LIN {X -196.784,Y -213.016,Z 123.751,A 47.268,B 90.000,C 0.000} C_DIS
LIN {X -197.620,Y -212.241,Z 123.582,A 47.043,B 90.000,C 0.000} C_DIS
LIN {X -198.410,Y -211.503,Z 123.560,A 46.829,B 90.000,C 0.000} C_DIS
LIN {X -199.108,Y -210.846,Z 123.719,A 46.640,B 90.000,C 0.000} C_DIS
LIN {X -199.675,Y -210.309,Z 123.966,A 46.486,B 90.000,C 0.000} C_DIS
LIN {X -200.147,Y -209.860,Z 124.319,A 46.357,B 90.000,C 0.000} C_DIS
LIN {X -200.558,Y -209.467,Z 124.798,A 46.245,B 90.000,C 0.000} C_DIS
LIN {X -200.980,Y -209.062,Z 125.590,A 46.129,B 90.000,C 0.000} C_DIS
LIN {X -201.312,Y -208.742,Z 126.725,A 46.038,B 90.000,C 0.000} C_DIS
LIN {X -201.468,Y -208.592,Z 127.575,A 45.995,B 90.000,C 0.000} C_DIS
LIN {X -201.547,Y -208.516,Z 128.408,A 45.974,B 90.000,C 0.000} C_DIS
LIN {X -201.548,Y -208.515,Z 129.167,A 45.973,B 90.000,C 0.000} C_DIS
LIN {X -201.440,Y -208.619,Z 130.066,A 46.003,B 90.000,C 0.000} C_DIS
LIN {X -201.835,Y -208.237,Z 129.890,A 45.895,B 90.000,C 0.000} C_DIS
LIN {X -202.884,Y -207.215,Z 129.170,A 45.605,B 90.000,C 0.000} C_DIS
LIN {X -204.304,Y -205.814,Z 127.663,A 45.211,B 90.000,C 0.000} C_DIS
LIN {X -204.732,Y -205.390,Z 127.194,A 45.092,B 90.000,C 0.000} C_DIS
LIN {X -205.294,Y -204.827,Z 126.844,A 44.935,B 90.000,C 0.000} C_DIS
LIN {X -206.113,Y -204.004,Z 126.614,A 44.705,B 90.000,C 0.000} C_DIS
LIN {X -207.863,Y -202.220,Z 126.527,A 44.212,B 90.000,C 0.000} C_DIS
LIN {X -207.932,Y -202.149,Z 126.529,A 44.192,B 90.000,C 0.000} C_DIS
LIN {X -208.601,Y -201.459,Z 126.690,A 44.002,B 90.000,C 0.000} C_DIS
LIN {X -208.848,Y -201.203,Z 126.861,A 43.932,B 90.000,C 0.000} C_DIS
LIN {X -209.068,Y -200.974,Z 127.141,A 43.869,B 90.000,C 0.000} C_DIS
LIN {X -209.459,Y -200.566,Z 128.088,A 43.757,B 90.000,C 0.000} C_DIS
LIN {X -209.762,Y -200.250,Z 129.265,A 43.671,B 90.000,C 0.000} C_DIS
LIN {X -209.850,Y -200.157,Z 130.407,A 43.646,B 90.000,C 0.000} C_DIS
LIN {X -209.802,Y -200.208,Z 131.716,A 43.659,B 90.000,C 0.000} C_DIS
LIN {X -209.567,Y -200.453,Z 132.873,A 43.727,B 90.000,C 0.000} C_DIS
LIN {X -209.190,Y -200.847,Z 134.012,A 43.834,B 90.000,C 0.000} C_DIS
LIN {X -207.748,Y -199.461,Z 134.012,A 43.834,B 90.000,C 0.000} C_DIS
WAIT SEC 0.1
RET=EKI_SetBool("oxy","torchState",FALSE)
RET = EKI_Send("oxy","torchState")
LIN {X -194.764,Y -186.995,Z 134.012,A 43.834,B 90.000,C 0.000} C_DIS
LIN {X -184.230,Y -197.381,Z 120.997,A 46.974,B 90.000,C 0.000} C_DIS
LIN {X -196.512,Y -210.540,Z 120.997,A 46.974,B 90.000,C 0.000} C_DIS
LIN {X -197.877,Y -212.002,Z 120.997,A 46.974,B 90.000,C 0.000} C_DIS
WAIT SEC 1
RET=EKI_SetBool("oxy","torchState",TRUE)
RET = EKI_Send("oxy","torchState")
LIN {X -198.195,Y -211.704,Z 120.444,A 46.888,B 90.000,C 0.000} C_DIS
LIN {X -198.412,Y -211.501,Z 119.734,A 46.829,B 90.000,C 0.000} C_DIS
LIN {X -198.488,Y -211.430,Z 117.237,A 46.808,B 90.000,C 0.000} C_DIS
LIN {X -198.366,Y -211.545,Z 115.557,A 46.841,B 90.000,C 0.000} C_DIS
LIN {X -198.150,Y -211.746,Z 114.873,A 46.900,B 90.000,C 0.000} C_DIS
LIN {X -197.024,Y -212.794,Z 112.902,A 47.204,B 90.000,C 0.000} C_DIS
LIN {X -196.854,Y -212.952,Z 112.641,A 47.249,B 90.000,C 0.000} C_DIS
LIN {X -196.638,Y -213.151,Z 112.446,A 47.308,B 90.000,C 0.000} C_DIS
LIN {X -196.433,Y -213.340,Z 112.465,A 47.363,B 90.000,C 0.000} C_DIS
LIN {X -196.193,Y -213.561,Z 112.727,A 47.427,B 90.000,C 0.000} C_DIS
LIN {X -195.388,Y -214.298,Z 113.920,A 47.643,B 90.000,C 0.000} C_DIS
LIN {X -193.851,Y -215.688,Z 115.318,A 48.052,B 90.000,C 0.000} C_DIS
LIN {X -192.222,Y -217.141,Z 116.537,A 48.483,B 90.000,C 0.000} C_DIS
LIN {X -190.581,Y -218.584,Z 117.751,A 48.915,B 90.000,C 0.000} C_DIS
LIN {X -189.444,Y -219.570,Z 118.907,A 49.213,B 90.000,C 0.000} C_DIS
LIN {X -188.072,Y -220.746,Z 120.635,A 49.570,B 90.000,C 0.000} C_DIS
LIN {X -186.854,Y -221.778,Z 122.333,A 49.885,B 90.000,C 0.000} C_DIS
LIN {X -186.543,Y -222.040,Z 123.009,A 49.965,B 90.000,C 0.000} C_DIS
LIN {X -186.357,Y -222.196,Z 123.639,A 50.013,B 90.000,C 0.000} C_DIS
LIN {X -186.301,Y -222.243,Z 124.194,A 50.028,B 90.000,C 0.000} C_DIS
LIN {X -186.382,Y -222.175,Z 124.643,A 50.007,B 90.000,C 0.000} C_DIS
LIN {X -186.558,Y -222.027,Z 124.964,A 49.961,B 90.000,C 0.000} C_DIS
LIN {X -186.818,Y -221.809,Z 125.228,A 49.894,B 90.000,C 0.000} C_DIS
LIN {X -187.628,Y -221.124,Z 125.617,A 49.685,B 90.000,C 0.000} C_DIS
LIN {X -189.526,Y -219.498,Z 125.677,A 49.191,B 90.000,C 0.000} C_DIS
LIN {X -189.856,Y -219.214,Z 125.662,A 49.105,B 90.000,C 0.000} C_DIS
LIN {X -190.574,Y -218.590,Z 125.514,A 48.917,B 90.000,C 0.000} C_DIS
LIN {X -191.225,Y -218.021,Z 125.214,A 48.746,B 90.000,C 0.000} C_DIS
LIN {X -192.885,Y -216.546,Z 124.065,A 48.308,B 90.000,C 0.000} C_DIS
LIN {X -194.538,Y -215.067,Z 122.914,A 47.869,B 90.000,C 0.000} C_DIS
LIN {X -194.792,Y -214.839,Z 122.737,A 47.802,B 90.000,C 0.000} C_DIS
LIN {X -196.523,Y -213.256,Z 121.874,A 47.338,B 90.000,C 0.000} C_DIS
LIN {X -197.278,Y -212.559,Z 121.499,A 47.135,B 90.000,C 0.000} C_DIS
LIN {X -197.877,Y -212.002,Z 120.997,A 46.974,B 90.000,C 0.000} C_DIS
LIN {X -196.512,Y -210.540,Z 120.997,A 46.974,B 90.000,C 0.000} C_DIS
WAIT SEC 0.1
RET=EKI_SetBool("oxy","torchState",FALSE)
RET = EKI_Send("oxy","torchState")
LIN {X -184.230,Y -197.381,Z 120.997,A 46.974,B 90.000,C 0.000} C_DIS
LIN {X -172.273,Y -207.899,Z 119.817,A 50.353,B 90.000,C 0.000} C_DIS
LIN {X -183.758,Y -221.759,Z 119.817,A 50.353,B 90.000,C 0.000} C_DIS
LIN {X -185.034,Y -223.299,Z 119.817,A 50.353,B 90.000,C 0.000} C_DIS
WAIT SEC 1
RET=EKI_SetBool("oxy","torchState",TRUE)
RET = EKI_Send("oxy","torchState")
LIN {X -184.856,Y -223.446,Z 120.126,A 50.399,B 90.000,C 0.000} C_DIS
LIN {X -183.667,Y -224.424,Z 121.180,A 50.703,B 90.000,C 0.000} C_DIS
LIN {X -183.201,Y -224.805,Z 121.693,A 50.822,B 90.000,C 0.000} C_DIS
LIN {X -182.861,Y -225.082,Z 122.228,A 50.909,B 90.000,C 0.000} C_DIS
LIN {X -182.593,Y -225.299,Z 122.854,A 50.977,B 90.000,C 0.000} C_DIS
LIN {X -182.365,Y -225.484,Z 123.690,A 51.035,B 90.000,C 0.000} C_DIS
LIN {X -182.269,Y -225.562,Z 124.538,A 51.060,B 90.000,C 0.000} C_DIS
LIN {X -182.306,Y -225.532,Z 125.372,A 51.050,B 90.000,C 0.000} C_DIS
LIN {X -182.478,Y -225.393,Z 126.167,A 51.006,B 90.000,C 0.000} C_DIS
LIN {X -182.602,Y -225.292,Z 126.492,A 50.975,B 90.000,C 0.000} C_DIS
LIN {X -182.769,Y -225.156,Z 126.725,A 50.932,B 90.000,C 0.000} C_DIS
LIN {X -184.097,Y -224.072,Z 127.477,A 50.593,B 90.000,C 0.000} C_DIS
LIN {X -184.322,Y -223.887,Z 127.745,A 50.536,B 90.000,C 0.000} C_DIS
LIN {X -184.356,Y -223.859,Z 127.968,A 50.527,B 90.000,C 0.000} C_DIS
LIN {X -184.259,Y -223.939,Z 128.176,A 50.552,B 90.000,C 0.000} C_DIS
LIN {X -183.010,Y -224.961,Z 129.049,A 50.871,B 90.000,C 0.000} C_DIS
LIN {X -182.638,Y -225.263,Z 129.597,A 50.966,B 90.000,C 0.000} C_DIS
LIN {X -182.380,Y -225.472,Z 130.408,A 51.031,B 90.000,C 0.000} C_DIS
LIN {X -182.249,Y -225.578,Z 131.423,A 51.065,B 90.000,C 0.000} C_DIS
LIN {X -182.257,Y -225.571,Z 132.585,A 51.062,B 90.000,C 0.000} C_DIS
LIN {X -182.405,Y -225.451,Z 133.925,A 51.025,B 90.000,C 0.000} C_DIS
LIN {X -182.958,Y -225.003,Z 136.321,A 50.884,B 90.000,C 0.000} C_DIS
LIN {X -183.203,Y -224.803,Z 137.226,A 50.822,B 90.000,C 0.000} C_DIS
LIN {X -183.718,Y -224.383,Z 138.429,A 50.690,B 90.000,C 0.000} C_DIS
LIN {X -184.128,Y -224.047,Z 139.041,A 50.586,B 90.000,C 0.000} C_DIS
LIN {X -185.312,Y -223.068,Z 140.256,A 50.282,B 90.000,C 0.000} C_DIS
LIN {X -185.472,Y -222.935,Z 140.613,A 50.241,B 90.000,C 0.000} C_DIS
LIN {X -185.325,Y -223.057,Z 140.910,A 50.279,B 90.000,C 0.000} C_DIS
LIN {X -183.861,Y -224.266,Z 142.531,A 50.654,B 90.000,C 0.000} C_DIS
LIN {X -183.152,Y -224.845,Z 143.576,A 50.835,B 90.000,C 0.000} C_DIS
LIN {X -182.817,Y -225.118,Z 144.247,A 50.920,B 90.000,C 0.000} C_DIS
LIN {X -182.642,Y -225.260,Z 144.909,A 50.965,B 90.000,C 0.000} C_DIS
LIN {X -182.537,Y -225.344,Z 145.889,A 50.991,B 90.000,C 0.000} C_DIS
LIN {X -182.508,Y -225.368,Z 148.389,A 50.999,B 90.000,C 0.000} C_DIS
LIN {X -182.531,Y -225.349,Z 150.889,A 50.993,B 90.000,C 0.000} C_DIS
LIN {X -182.593,Y -225.299,Z 153.021,A 50.977,B 90.000,C 0.000} C_DIS
LIN {X -182.731,Y -225.188,Z 154.059,A 50.942,B 90.000,C 0.000} C_DIS
LIN {X -183.254,Y -224.762,Z 156.466,A 50.809,B 90.000,C 0.000} C_DIS
LIN {X -183.583,Y -224.493,Z 158.013,A 50.725,B 90.000,C 0.000} C_DIS
LIN {X -184.559,Y -223.690,Z 160.170,A 50.475,B 90.000,C 0.000} C_DIS
LIN {X -185.518,Y -222.897,Z 162.338,A 50.229,B 90.000,C 0.000} C_DIS
LIN {X -186.373,Y -222.181,Z 164.576,A 50.009,B 90.000,C 0.000} C_DIS
LIN {X -187.164,Y -221.516,Z 166.852,A 49.805,B 90.000,C 0.000} C_DIS
LIN {X -187.859,Y -220.927,Z 169.180,A 49.625,B 90.000,C 0.000} C_DIS
LIN {X -188.439,Y -220.433,Z 171.561,A 49.474,B 90.000,C 0.000} C_DIS
LIN {X -188.491,Y -220.389,Z 171.776,A 49.461,B 90.000,C 0.000} C_DIS
LIN {X -188.839,Y -220.090,Z 174.234,A 49.370,B 90.000,C 0.000} C_DIS
LIN {X -189.057,Y -219.903,Z 176.717,A 49.313,B 90.000,C 0.000} C_DIS
LIN {X -189.184,Y -219.794,Z 179.211,A 49.280,B 90.000,C 0.000} C_DIS
LIN {X -189.234,Y -219.751,Z 181.710,A 49.267,B 90.000,C 0.000} C_DIS
LIN {X -189.219,Y -219.764,Z 184.210,A 49.271,B 90.000,C 0.000} C_DIS
LIN {X -189.133,Y -219.837,Z 186.708,A 49.294,B 90.000,C 0.000} C_DIS
LIN {X -188.954,Y -219.992,Z 189.196,A 49.340,B 90.000,C 0.000} C_DIS
LIN {X -188.655,Y -220.248,Z 191.665,A 49.418,B 90.000,C 0.000} C_DIS
LIN {X -188.211,Y -220.627,Z 194.096,A 49.533,B 90.000,C 0.000} C_DIS
LIN {X -187.648,Y -221.106,Z 196.484,A 49.679,B 90.000,C 0.000} C_DIS
LIN {X -186.944,Y -221.702,Z 198.808,A 49.862,B 90.000,C 0.000} C_DIS
LIN {X -186.113,Y -222.400,Z 201.059,A 50.076,B 90.000,C 0.000} C_DIS
LIN {X -185.249,Y -223.121,Z 203.042,A 50.298,B 90.000,C 0.000} C_DIS
LIN {X -184.688,Y -223.585,Z 203.997,A 50.442,B 90.000,C 0.000} C_DIS
LIN {X -184.135,Y -224.041,Z 204.652,A 50.584,B 90.000,C 0.000} C_DIS
LIN {X -183.571,Y -224.503,Z 205.036,A 50.728,B 90.000,C 0.000} C_DIS
LIN {X -182.939,Y -225.018,Z 205.136,A 50.889,B 90.000,C 0.000} C_DIS
LIN {X -182.361,Y -225.487,Z 205.050,A 51.036,B 90.000,C 0.000} C_DIS
LIN {X -182.219,Y -225.602,Z 204.969,A 51.072,B 90.000,C 0.000} C_DIS
LIN {X -183.025,Y -224.948,Z 202.695,A 50.867,B 90.000,C 0.000} C_DIS
LIN {X -183.743,Y -224.362,Z 200.373,A 50.684,B 90.000,C 0.000} C_DIS
LIN {X -183.893,Y -224.240,Z 199.868,A 50.646,B 90.000,C 0.000} C_DIS
LIN {X -184.233,Y -223.960,Z 197.407,A 50.559,B 90.000,C 0.000} C_DIS
LIN {X -184.543,Y -223.705,Z 194.940,A 50.479,B 90.000,C 0.000} C_DIS
LIN {X -184.839,Y -223.460,Z 192.470,A 50.404,B 90.000,C 0.000} C_DIS
LIN {X -184.845,Y -223.456,Z 192.407,A 50.402,B 90.000,C 0.000} C_DIS
LIN {X -184.845,Y -223.455,Z 189.907,A 50.402,B 90.000,C 0.000} C_DIS
LIN {X -184.775,Y -223.513,Z 187.734,A 50.420,B 90.000,C 0.000} C_DIS
LIN {X -184.612,Y -223.648,Z 186.808,A 50.462,B 90.000,C 0.000} C_DIS
LIN {X -183.782,Y -224.330,Z 184.550,A 50.674,B 90.000,C 0.000} C_DIS
LIN {X -183.366,Y -224.671,Z 183.534,A 50.780,B 90.000,C 0.000} C_DIS
LIN {X -182.026,Y -225.757,Z 181.725,A 51.121,B 90.000,C 0.000} C_DIS
LIN {X -181.496,Y -226.184,Z 181.032,A 51.256,B 90.000,C 0.000} C_DIS
LIN {X -180.136,Y -227.267,Z 182.829,A 51.599,B 90.000,C 0.000} C_DIS
LIN {X -179.786,Y -227.545,Z 183.304,A 51.687,B 90.000,C 0.000} C_DIS
LIN {X -178.829,Y -228.298,Z 185.487,A 51.928,B 90.000,C 0.000} C_DIS
LIN {X -178.303,Y -228.710,Z 186.994,A 52.060,B 90.000,C 0.000} C_DIS
LIN {X -178.184,Y -228.802,Z 187.723,A 52.090,B 90.000,C 0.000} C_DIS
LIN {X -178.074,Y -228.888,Z 190.219,A 52.117,B 90.000,C 0.000} C_DIS
LIN {X -178.030,Y -228.922,Z 191.004,A 52.128,B 90.000,C 0.000} C_DIS
LIN {X -178.185,Y -228.801,Z 193.496,A 52.089,B 90.000,C 0.000} C_DIS
LIN {X -178.597,Y -228.480,Z 195.941,A 51.986,B 90.000,C 0.000} C_DIS
LIN {X -178.860,Y -228.274,Z 198.418,A 51.920,B 90.000,C 0.000} C_DIS
LIN {X -178.906,Y -228.238,Z 198.848,A 51.909,B 90.000,C 0.000} C_DIS
LIN {X -179.424,Y -227.831,Z 201.260,A 51.778,B 90.000,C 0.000} C_DIS
LIN {X -179.461,Y -227.802,Z 201.420,A 51.769,B 90.000,C 0.000} C_DIS
LIN {X -180.303,Y -227.136,Z 203.678,A 51.557,B 90.000,C 0.000} C_DIS
LIN {X -180.796,Y -226.744,Z 205.012,A 51.433,B 90.000,C 0.000} C_DIS
LIN {X -180.725,Y -226.801,Z 205.094,A 51.451,B 90.000,C 0.000} C_DIS
LIN {X -179.824,Y -227.515,Z 205.070,A 51.678,B 90.000,C 0.000} C_DIS
LIN {X -179.385,Y -227.862,Z 204.925,A 51.788,B 90.000,C 0.000} C_DIS
LIN {X -179.000,Y -228.165,Z 204.647,A 51.885,B 90.000,C 0.000} C_DIS
LIN {X -178.608,Y -228.472,Z 204.205,A 51.983,B 90.000,C 0.000} C_DIS
LIN {X -178.121,Y -228.851,Z 203.462,A 52.105,B 90.000,C 0.000} C_DIS
LIN {X -177.146,Y -229.605,Z 201.287,A 52.349,B 90.000,C 0.000} C_DIS
LIN {X -176.254,Y -230.291,Z 199.055,A 52.571,B 90.000,C 0.000} C_DIS
LIN {X -175.456,Y -230.901,Z 196.766,A 52.770,B 90.000,C 0.000} C_DIS
LIN {X -175.320,Y -231.004,Z 196.344,A 52.804,B 90.000,C 0.000} C_DIS
LIN {X -174.777,Y -231.415,Z 193.939,A 52.938,B 90.000,C 0.000} C_DIS
LIN {X -174.334,Y -231.749,Z 191.501,A 53.048,B 90.000,C 0.000} C_DIS
LIN {X -173.993,Y -232.005,Z 189.038,A 53.132,B 90.000,C 0.000} C_DIS
LIN {X -173.793,Y -232.155,Z 186.551,A 53.181,B 90.000,C 0.000} C_DIS
LIN {X -173.712,Y -232.216,Z 184.053,A 53.201,B 90.000,C 0.000} C_DIS
LIN {X -173.713,Y -232.215,Z 181.553,A 53.201,B 90.000,C 0.000} C_DIS
LIN {X -173.765,Y -232.176,Z 179.054,A 53.188,B 90.000,C 0.000} C_DIS
LIN {X -173.905,Y -232.071,Z 176.560,A 53.153,B 90.000,C 0.000} C_DIS
LIN {X -174.167,Y -231.874,Z 174.082,A 53.089,B 90.000,C 0.000} C_DIS
LIN {X -174.556,Y -231.582,Z 171.630,A 52.993,B 90.000,C 0.000} C_DIS
LIN {X -174.754,Y -231.433,Z 170.547,A 52.944,B 90.000,C 0.000} C_DIS
LIN {X -175.428,Y -230.922,Z 168.195,A 52.777,B 90.000,C 0.000} C_DIS
LIN {X -176.255,Y -230.289,Z 165.922,A 52.571,B 90.000,C 0.000} C_DIS
LIN {X -177.099,Y -229.643,Z 163.659,A 52.361,B 90.000,C 0.000} C_DIS
LIN {X -177.978,Y -228.963,Z 161.420,A 52.141,B 90.000,C 0.000} C_DIS
LIN {X -179.007,Y -228.159,Z 159.288,A 51.883,B 90.000,C 0.000} C_DIS
LIN {X -179.501,Y -227.770,Z 158.263,A 51.759,B 90.000,C 0.000} C_DIS
LIN {X -180.062,Y -227.327,Z 155.868,A 51.618,B 90.000,C 0.000} C_DIS
LIN {X -180.524,Y -226.960,Z 153.438,A 51.501,B 90.000,C 0.000} C_DIS
LIN {X -180.619,Y -226.885,Z 152.682,A 51.477,B 90.000,C 0.000} C_DIS
LIN {X -180.685,Y -226.832,Z 150.183,A 51.461,B 90.000,C 0.000} C_DIS
LIN {X -180.683,Y -226.834,Z 147.683,A 51.461,B 90.000,C 0.000} C_DIS
LIN {X -180.639,Y -226.869,Z 145.712,A 51.472,B 90.000,C 0.000} C_DIS
LIN {X -180.427,Y -227.038,Z 144.468,A 51.526,B 90.000,C 0.000} C_DIS
LIN {X -179.559,Y -227.725,Z 142.753,A 51.745,B 90.000,C 0.000} C_DIS
LIN {X -179.064,Y -228.114,Z 142.087,A 51.869,B 90.000,C 0.000} C_DIS
LIN {X -177.715,Y -229.167,Z 140.827,A 52.207,B 90.000,C 0.000} C_DIS
LIN {X -177.642,Y -229.223,Z 140.536,A 52.225,B 90.000,C 0.000} C_DIS
LIN {X -178.714,Y -228.389,Z 139.353,A 51.957,B 90.000,C 0.000} C_DIS
LIN {X -179.237,Y -227.978,Z 138.656,A 51.825,B 90.000,C 0.000} C_DIS
LIN {X -179.676,Y -227.632,Z 137.918,A 51.715,B 90.000,C 0.000} C_DIS
LIN {X -180.022,Y -227.359,Z 137.149,A 51.628,B 90.000,C 0.000} C_DIS
LIN {X -180.593,Y -226.906,Z 134.757,A 51.484,B 90.000,C 0.000} C_DIS
LIN {X -180.917,Y -226.648,Z 132.791,A 51.402,B 90.000,C 0.000} C_DIS
LIN {X -180.971,Y -226.605,Z 131.507,A 51.388,B 90.000,C 0.000} C_DIS
LIN {X -180.866,Y -226.688,Z 130.430,A 51.415,B 90.000,C 0.000} C_DIS
LIN {X -180.603,Y -226.897,Z 129.631,A 51.481,B 90.000,C 0.000} C_DIS
LIN {X -180.163,Y -227.247,Z 129.064,A 51.592,B 90.000,C 0.000} C_DIS
LIN {X -178.919,Y -228.228,Z 128.205,A 51.905,B 90.000,C 0.000} C_DIS
LIN {X -178.801,Y -228.321,Z 127.998,A 51.935,B 90.000,C 0.000} C_DIS
LIN {X -178.815,Y -228.310,Z 127.787,A 51.932,B 90.000,C 0.000} C_DIS
LIN {X -178.955,Y -228.200,Z 127.588,A 51.896,B 90.000,C 0.000} C_DIS
LIN {X -180.272,Y -227.161,Z 126.826,A 51.565,B 90.000,C 0.000} C_DIS
LIN {X -180.540,Y -226.948,Z 126.548,A 51.497,B 90.000,C 0.000} C_DIS
LIN {X -180.705,Y -226.816,Z 126.225,A 51.456,B 90.000,C 0.000} C_DIS
LIN {X -180.889,Y -226.670,Z 125.437,A 51.409,B 90.000,C 0.000} C_DIS
LIN {X -180.917,Y -226.648,Z 124.452,A 51.402,B 90.000,C 0.000} C_DIS
LIN {X -180.857,Y -226.696,Z 123.746,A 51.417,B 90.000,C 0.000} C_DIS
LIN {X -180.732,Y -226.795,Z 123.144,A 51.449,B 90.000,C 0.000} C_DIS
LIN {X -180.530,Y -226.956,Z 122.604,A 51.500,B 90.000,C 0.000} C_DIS
LIN {X -180.239,Y -227.187,Z 122.083,A 51.573,B 90.000,C 0.000} C_DIS
LIN {X -179.700,Y -227.613,Z 121.403,A 51.709,B 90.000,C 0.000} C_DIS
LIN {X -178.128,Y -228.846,Z 119.900,A 52.104,B 90.000,C 0.000} C_DIS
LIN {X -178.358,Y -228.667,Z 119.465,A 52.046,B 90.000,C 0.000} C_DIS
LIN {X -179.811,Y -227.526,Z 117.832,A 51.681,B 90.000,C 0.000} C_DIS
LIN {X -180.037,Y -227.347,Z 117.382,A 51.624,B 90.000,C 0.000} C_DIS
LIN {X -180.191,Y -227.225,Z 116.862,A 51.585,B 90.000,C 0.000} C_DIS
LIN {X -180.352,Y -227.097,Z 115.826,A 51.545,B 90.000,C 0.000} C_DIS
LIN {X -180.401,Y -227.058,Z 114.729,A 51.532,B 90.000,C 0.000} C_DIS
LIN {X -180.339,Y -227.108,Z 113.721,A 51.548,B 90.000,C 0.000} C_DIS
LIN {X -180.166,Y -227.245,Z 112.951,A 51.592,B 90.000,C 0.000} C_DIS
LIN {X -179.769,Y -227.559,Z 112.193,A 51.692,B 90.000,C 0.000} C_DIS
LIN {X -179.172,Y -228.029,Z 111.327,A 51.842,B 90.000,C 0.000} C_DIS
LIN {X -178.806,Y -228.316,Z 110.909,A 51.934,B 90.000,C 0.000} C_DIS
LIN {X -177.696,Y -229.181,Z 110.174,A 52.212,B 90.000,C 0.000} C_DIS
LIN {X -177.428,Y -229.389,Z 109.917,A 52.279,B 90.000,C 0.000} C_DIS
LIN {X -177.359,Y -229.443,Z 109.721,A 52.296,B 90.000,C 0.000} C_DIS
LIN {X -177.405,Y -229.407,Z 109.491,A 52.284,B 90.000,C 0.000} C_DIS
LIN {X -178.685,Y -228.411,Z 107.589,A 51.964,B 90.000,C 0.000} C_DIS
LIN {X -178.907,Y -228.237,Z 107.259,A 51.908,B 90.000,C 0.000} C_DIS
LIN {X -179.983,Y -227.390,Z 105.167,A 51.638,B 90.000,C 0.000} C_DIS
LIN {X -181.072,Y -226.523,Z 103.091,A 51.363,B 90.000,C 0.000} C_DIS
LIN {X -181.391,Y -226.268,Z 102.518,A 51.282,B 90.000,C 0.000} C_DIS
LIN {X -181.572,Y -226.123,Z 102.429,A 51.236,B 90.000,C 0.000} C_DIS
LIN {X -181.773,Y -225.961,Z 102.518,A 51.185,B 90.000,C 0.000} C_DIS
LIN {X -182.096,Y -225.701,Z 102.964,A 51.103,B 90.000,C 0.000} C_DIS
LIN {X -183.137,Y -224.856,Z 105.075,A 50.839,B 90.000,C 0.000} C_DIS
LIN {X -183.971,Y -224.175,Z 106.720,A 50.626,B 90.000,C 0.000} C_DIS
LIN {X -185.205,Y -223.156,Z 108.640,A 50.309,B 90.000,C 0.000} C_DIS
LIN {X -185.718,Y -222.730,Z 109.444,A 50.178,B 90.000,C 0.000} C_DIS
LIN {X -185.765,Y -222.691,Z 109.795,A 50.166,B 90.000,C 0.000} C_DIS
LIN {X -185.521,Y -222.894,Z 110.114,A 50.228,B 90.000,C 0.000} C_DIS
LIN {X -184.442,Y -223.788,Z 110.864,A 50.505,B 90.000,C 0.000} C_DIS
LIN {X -184.036,Y -224.122,Z 111.307,A 50.609,B 90.000,C 0.000} C_DIS
LIN {X -183.409,Y -224.636,Z 112.183,A 50.769,B 90.000,C 0.000} C_DIS
LIN {X -183.025,Y -224.948,Z 112.920,A 50.867,B 90.000,C 0.000} C_DIS
LIN {X -182.832,Y -225.106,Z 113.909,A 50.916,B 90.000,C 0.000} C_DIS
LIN {X -182.794,Y -225.137,Z 115.170,A 50.926,B 90.000,C 0.000} C_DIS
LIN {X -182.903,Y -225.048,Z 116.440,A 50.898,B 90.000,C 0.000} C_DIS
LIN {X -183.153,Y -224.844,Z 117.457,A 50.835,B 90.000,C 0.000} C_DIS
LIN {X -183.510,Y -224.553,Z 118.037,A 50.744,B 90.000,C 0.000} C_DIS
LIN {X -184.851,Y -223.450,Z 119.459,A 50.400,B 90.000,C 0.000} C_DIS
LIN {X -185.034,Y -223.299,Z 119.817,A 50.353,B 90.000,C 0.000} C_DIS
LIN {X -183.758,Y -221.759,Z 119.817,A 50.353,B 90.000,C 0.000} C_DIS
WAIT SEC 0.1
RET=EKI_SetBool("oxy","torchState",FALSE)
RET = EKI_Send("oxy","torchState")
LIN {X -172.273,Y -207.899,Z 119.817,A 50.353,B 90.000,C 0.000} C_DIS
LIN {X -164.615,Y -214.014,Z 123.791,A 52.433,B 90.000,C 0.000} C_DIS
LIN {X -175.589,Y -228.281,Z 123.791,A 52.433,B 90.000,C 0.000} C_DIS
LIN {X -176.809,Y -229.867,Z 123.791,A 52.433,B 90.000,C 0.000} C_DIS
WAIT SEC 1
RET=EKI_SetBool("oxy","torchState",TRUE)
RET = EKI_Send("oxy","torchState")
LIN {X -176.854,Y -229.831,Z 124.177,A 52.422,B 90.000,C 0.000} C_DIS
LIN {X -176.773,Y -229.894,Z 124.634,A 52.442,B 90.000,C 0.000} C_DIS
LIN {X -176.531,Y -230.080,Z 125.022,A 52.502,B 90.000,C 0.000} C_DIS
LIN {X -176.132,Y -230.385,Z 125.338,A 52.602,B 90.000,C 0.000} C_DIS
LIN {X -175.578,Y -230.808,Z 125.577,A 52.739,B 90.000,C 0.000} C_DIS
LIN {X -174.415,Y -231.688,Z 125.727,A 53.027,B 90.000,C 0.000} C_DIS
LIN {X -173.083,Y -232.685,Z 125.688,A 53.356,B 90.000,C 0.000} C_DIS
LIN {X -172.414,Y -233.181,Z 125.564,A 53.521,B 90.000,C 0.000} C_DIS
LIN {X -171.862,Y -233.588,Z 125.378,A 53.656,B 90.000,C 0.000} C_DIS
LIN {X -171.338,Y -233.973,Z 125.091,A 53.785,B 90.000,C 0.000} C_DIS
LIN {X -169.585,Y -235.245,Z 123.843,A 54.213,B 90.000,C 0.000} C_DIS
LIN {X -167.767,Y -236.546,Z 122.723,A 54.654,B 90.000,C 0.000} C_DIS
LIN {X -165.840,Y -237.901,Z 121.888,A 55.120,B 90.000,C 0.000} C_DIS
LIN {X -164.814,Y -238.613,Z 121.431,A 55.367,B 90.000,C 0.000} C_DIS
LIN {X -164.408,Y -238.893,Z 121.131,A 55.464,B 90.000,C 0.000} C_DIS
LIN {X -164.103,Y -239.103,Z 120.775,A 55.537,B 90.000,C 0.000} C_DIS
LIN {X -163.884,Y -239.253,Z 120.342,A 55.590,B 90.000,C 0.000} C_DIS
LIN {X -163.738,Y -239.353,Z 119.812,A 55.625,B 90.000,C 0.000} C_DIS
LIN {X -163.608,Y -239.442,Z 118.373,A 55.656,B 90.000,C 0.000} C_DIS
LIN {X -163.677,Y -239.394,Z 116.274,A 55.639,B 90.000,C 0.000} C_DIS
LIN {X -163.813,Y -239.302,Z 115.449,A 55.607,B 90.000,C 0.000} C_DIS
LIN {X -164.014,Y -239.164,Z 114.789,A 55.558,B 90.000,C 0.000} C_DIS
LIN {X -165.309,Y -238.270,Z 112.846,A 55.248,B 90.000,C 0.000} C_DIS
LIN {X -165.460,Y -238.166,Z 112.641,A 55.211,B 90.000,C 0.000} C_DIS
LIN {X -165.794,Y -237.934,Z 112.428,A 55.131,B 90.000,C 0.000} C_DIS
LIN {X -166.128,Y -237.701,Z 112.641,A 55.051,B 90.000,C 0.000} C_DIS
LIN {X -167.164,Y -236.973,Z 113.994,A 54.800,B 90.000,C 0.000} C_DIS
LIN {X -168.853,Y -235.770,Z 115.391,A 54.391,B 90.000,C 0.000} C_DIS
LIN {X -170.616,Y -234.497,Z 116.625,A 53.961,B 90.000,C 0.000} C_DIS
LIN {X -172.371,Y -233.212,Z 117.856,A 53.531,B 90.000,C 0.000} C_DIS
LIN {X -172.777,Y -232.912,Z 118.163,A 53.432,B 90.000,C 0.000} C_DIS
LIN {X -174.273,Y -231.795,Z 119.825,A 53.063,B 90.000,C 0.000} C_DIS
LIN {X -175.685,Y -230.726,Z 121.589,A 52.713,B 90.000,C 0.000} C_DIS
LIN {X -176.089,Y -230.419,Z 122.185,A 52.612,B 90.000,C 0.000} C_DIS
LIN {X -176.669,Y -229.974,Z 123.338,A 52.468,B 90.000,C 0.000} C_DIS
LIN {X -176.809,Y -229.867,Z 123.791,A 52.433,B 90.000,C 0.000} C_DIS
LIN {X -175.589,Y -228.281,Z 123.791,A 52.433,B 90.000,C 0.000} C_DIS
WAIT SEC 0.1
RET=EKI_SetBool("oxy","torchState",FALSE)
RET = EKI_Send("oxy","torchState")
LIN {X -164.615,Y -214.014,Z 123.791,A 52.433,B 90.000,C 0.000} C_DIS
LIN {X -163.913,Y -214.552,Z 127.340,A 52.621,B 90.000,C 0.000} C_DIS
LIN {X -174.841,Y -228.855,Z 127.340,A 52.621,B 90.000,C 0.000} C_DIS
LIN {X -176.055,Y -230.444,Z 127.340,A 52.621,B 90.000,C 0.000} C_DIS
WAIT SEC 1
RET=EKI_SetBool("oxy","torchState",TRUE)
RET = EKI_Send("oxy","torchState")
LIN {X -175.617,Y -230.779,Z 126.995,A 52.730,B 90.000,C 0.000} C_DIS
LIN {X -175.023,Y -231.229,Z 126.772,A 52.877,B 90.000,C 0.000} C_DIS
LIN {X -174.268,Y -231.799,Z 126.669,A 53.064,B 90.000,C 0.000} C_DIS
LIN {X -173.368,Y -232.473,Z 126.693,A 53.286,B 90.000,C 0.000} C_DIS
LIN {X -172.541,Y -233.087,Z 126.886,A 53.490,B 90.000,C 0.000} C_DIS
LIN {X -171.801,Y -233.633,Z 127.250,A 53.671,B 90.000,C 0.000} C_DIS
LIN {X -170.250,Y -234.766,Z 128.851,A 54.051,B 90.000,C 0.000} C_DIS
LIN {X -170.203,Y -234.800,Z 128.901,A 54.062,B 90.000,C 0.000} C_DIS
LIN {X -169.403,Y -235.377,Z 129.534,A 54.257,B 90.000,C 0.000} C_DIS
LIN {X -169.110,Y -235.588,Z 129.714,A 54.328,B 90.000,C 0.000} C_DIS
LIN {X -168.972,Y -235.688,Z 129.701,A 54.362,B 90.000,C 0.000} C_DIS
LIN {X -168.908,Y -235.733,Z 127.707,A 54.378,B 90.000,C 0.000} C_DIS
LIN {X -168.826,Y -235.792,Z 127.150,A 54.398,B 90.000,C 0.000} C_DIS
LIN {X -168.563,Y -235.980,Z 126.231,A 54.461,B 90.000,C 0.000} C_DIS
LIN {X -168.230,Y -236.217,Z 125.496,A 54.542,B 90.000,C 0.000} C_DIS
LIN {X -167.822,Y -236.508,Z 124.935,A 54.641,B 90.000,C 0.000} C_DIS
LIN {X -167.331,Y -236.855,Z 124.539,A 54.760,B 90.000,C 0.000} C_DIS
LIN {X -166.224,Y -237.633,Z 124.015,A 55.027,B 90.000,C 0.000} C_DIS
LIN {X -165.003,Y -238.483,Z 123.663,A 55.321,B 90.000,C 0.000} C_DIS
LIN {X -165.003,Y -238.483,Z 123.663,A 55.321,B 90.000,C 0.000} C_DIS
LIN {X -163.875,Y -239.259,Z 123.604,A 55.592,B 90.000,C 0.000} C_DIS
LIN {X -162.859,Y -239.952,Z 123.723,A 55.835,B 90.000,C 0.000} C_DIS
LIN {X -162.012,Y -240.525,Z 124.092,A 56.037,B 90.000,C 0.000} C_DIS
LIN {X -161.434,Y -240.913,Z 124.565,A 56.174,B 90.000,C 0.000} C_DIS
LIN {X -160.949,Y -241.237,Z 125.264,A 56.289,B 90.000,C 0.000} C_DIS
LIN {X -160.552,Y -241.502,Z 126.200,A 56.384,B 90.000,C 0.000} C_DIS
LIN {X -160.236,Y -241.712,Z 127.384,A 56.459,B 90.000,C 0.000} C_DIS
LIN {X -160.103,Y -241.800,Z 128.427,A 56.490,B 90.000,C 0.000} C_DIS
LIN {X -160.224,Y -241.719,Z 130.106,A 56.462,B 90.000,C 0.000} C_DIS
LIN {X -159.105,Y -242.457,Z 129.527,A 56.726,B 90.000,C 0.000} C_DIS
LIN {X -158.128,Y -243.096,Z 128.840,A 56.957,B 90.000,C 0.000} C_DIS
LIN {X -156.485,Y -244.156,Z 127.282,A 57.343,B 90.000,C 0.000} C_DIS
LIN {X -156.451,Y -244.178,Z 127.249,A 57.351,B 90.000,C 0.000} C_DIS
LIN {X -155.901,Y -244.530,Z 126.902,A 57.480,B 90.000,C 0.000} C_DIS
LIN {X -154.390,Y -245.487,Z 126.605,A 57.834,B 90.000,C 0.000} C_DIS
LIN {X -152.601,Y -246.603,Z 126.496,A 58.250,B 90.000,C 0.000} C_DIS
LIN {X -151.725,Y -247.143,Z 126.634,A 58.454,B 90.000,C 0.000} C_DIS
LIN {X -151.435,Y -247.321,Z 126.797,A 58.521,B 90.000,C 0.000} C_DIS
LIN {X -151.177,Y -247.478,Z 127.049,A 58.581,B 90.000,C 0.000} C_DIS
LIN {X -150.759,Y -247.733,Z 127.754,A 58.677,B 90.000,C 0.000} C_DIS
LIN {X -150.395,Y -247.954,Z 128.700,A 58.761,B 90.000,C 0.000} C_DIS
LIN {X -150.174,Y -248.088,Z 129.900,A 58.812,B 90.000,C 0.000} C_DIS
LIN {X -150.183,Y -248.083,Z 131.171,A 58.810,B 90.000,C 0.000} C_DIS
LIN {X -150.420,Y -247.939,Z 132.490,A 58.756,B 90.000,C 0.000} C_DIS
LIN {X -150.882,Y -247.658,Z 133.834,A 58.649,B 90.000,C 0.000} C_DIS
LIN {X -151.417,Y -247.332,Z 134.926,A 58.525,B 90.000,C 0.000} C_DIS
LIN {X -152.064,Y -246.934,Z 135.854,A 58.375,B 90.000,C 0.000} C_DIS
LIN {X -153.715,Y -245.909,Z 137.426,A 57.991,B 90.000,C 0.000} C_DIS
LIN {X -154.917,Y -245.155,Z 138.488,A 57.711,B 90.000,C 0.000} C_DIS
LIN {X -155.512,Y -244.778,Z 139.171,A 57.571,B 90.000,C 0.000} C_DIS
LIN {X -156.005,Y -244.464,Z 139.903,A 57.456,B 90.000,C 0.000} C_DIS
LIN {X -156.392,Y -244.216,Z 140.677,A 57.365,B 90.000,C 0.000} C_DIS
LIN {X -156.888,Y -243.898,Z 142.233,A 57.249,B 90.000,C 0.000} C_DIS
LIN {X -157.178,Y -243.711,Z 142.477,A 57.181,B 90.000,C 0.000} C_DIS
LIN {X -157.583,Y -243.449,Z 142.582,A 57.085,B 90.000,C 0.000} C_DIS
LIN {X -157.993,Y -243.184,Z 142.504,A 56.989,B 90.000,C 0.000} C_DIS
LIN {X -158.525,Y -242.837,Z 142.281,A 56.863,B 90.000,C 0.000} C_DIS
LIN {X -160.378,Y -241.617,Z 141.130,A 56.425,B 90.000,C 0.000} C_DIS
LIN {X -160.602,Y -241.468,Z 140.995,A 56.372,B 90.000,C 0.000} C_DIS
LIN {X -160.898,Y -241.271,Z 140.926,A 56.302,B 90.000,C 0.000} C_DIS
LIN {X -161.117,Y -241.125,Z 140.973,A 56.250,B 90.000,C 0.000} C_DIS
LIN {X -161.260,Y -241.030,Z 141.137,A 56.216,B 90.000,C 0.000} C_DIS
LIN {X -161.324,Y -240.987,Z 141.416,A 56.200,B 90.000,C 0.000} C_DIS
LIN {X -161.213,Y -241.061,Z 142.319,A 56.227,B 90.000,C 0.000} C_DIS
LIN {X -160.983,Y -241.214,Z 143.095,A 56.281,B 90.000,C 0.000} C_DIS
LIN {X -160.675,Y -241.420,Z 143.698,A 56.355,B 90.000,C 0.000} C_DIS
LIN {X -160.204,Y -241.733,Z 144.249,A 56.466,B 90.000,C 0.000} C_DIS
LIN {X -158.453,Y -242.884,Z 145.613,A 56.880,B 90.000,C 0.000} C_DIS
LIN {X -158.418,Y -242.907,Z 145.638,A 56.889,B 90.000,C 0.000} C_DIS
LIN {X -158.037,Y -243.155,Z 145.746,A 56.978,B 90.000,C 0.000} C_DIS
LIN {X -155.937,Y -244.507,Z 145.646,A 57.472,B 90.000,C 0.000} C_DIS
LIN {X -154.610,Y -245.348,Z 145.553,A 57.782,B 90.000,C 0.000} C_DIS
LIN {X -154.152,Y -245.636,Z 145.627,A 57.889,B 90.000,C 0.000} C_DIS
LIN {X -153.760,Y -245.882,Z 145.791,A 57.981,B 90.000,C 0.000} C_DIS
LIN {X -153.319,Y -246.157,Z 146.147,A 58.083,B 90.000,C 0.000} C_DIS
LIN {X -153.020,Y -246.343,Z 146.670,A 58.153,B 90.000,C 0.000} C_DIS
LIN {X -152.858,Y -246.444,Z 147.374,A 58.191,B 90.000,C 0.000} C_DIS
LIN {X -152.828,Y -246.462,Z 148.268,A 58.198,B 90.000,C 0.000} C_DIS
LIN {X -152.940,Y -246.393,Z 149.090,A 58.171,B 90.000,C 0.000} C_DIS
LIN {X -153.297,Y -246.171,Z 149.656,A 58.088,B 90.000,C 0.000} C_DIS
LIN {X -153.665,Y -245.941,Z 149.988,A 58.003,B 90.000,C 0.000} C_DIS
LIN {X -154.087,Y -245.677,Z 150.199,A 57.904,B 90.000,C 0.000} C_DIS
LIN {X -154.627,Y -245.337,Z 150.309,A 57.778,B 90.000,C 0.000} C_DIS
LIN {X -155.349,Y -244.881,Z 150.342,A 57.610,B 90.000,C 0.000} C_DIS
LIN {X -156.653,Y -244.049,Z 150.234,A 57.304,B 90.000,C 0.000} C_DIS
LIN {X -157.762,Y -243.333,Z 149.889,A 57.043,B 90.000,C 0.000} C_DIS
LIN {X -158.734,Y -242.701,Z 149.282,A 56.814,B 90.000,C 0.000} C_DIS
LIN {X -159.625,Y -242.116,Z 148.387,A 56.603,B 90.000,C 0.000} C_DIS
LIN {X -160.172,Y -241.754,Z 147.654,A 56.474,B 90.000,C 0.000} C_DIS
LIN {X -160.685,Y -241.413,Z 146.787,A 56.352,B 90.000,C 0.000} C_DIS
LIN {X -161.675,Y -240.751,Z 144.589,A 56.117,B 90.000,C 0.000} C_DIS
LIN {X -162.561,Y -240.153,Z 142.329,A 55.906,B 90.000,C 0.000} C_DIS
LIN {X -162.701,Y -240.059,Z 141.961,A 55.872,B 90.000,C 0.000} C_DIS
LIN {X -163.364,Y -239.608,Z 139.593,A 55.714,B 90.000,C 0.000} C_DIS
LIN {X -163.415,Y -239.574,Z 139.431,A 55.702,B 90.000,C 0.000} C_DIS
LIN {X -163.658,Y -239.408,Z 139.065,A 55.644,B 90.000,C 0.000} C_DIS
LIN {X -165.346,Y -238.243,Z 137.636,A 55.238,B 90.000,C 0.000} C_DIS
LIN {X -167.101,Y -237.017,Z 136.345,A 54.815,B 90.000,C 0.000} C_DIS
LIN {X -168.872,Y -235.758,Z 135.109,A 54.386,B 90.000,C 0.000} C_DIS
LIN {X -169.485,Y -235.318,Z 134.700,A 54.237,B 90.000,C 0.000} C_DIS
LIN {X -170.054,Y -234.907,Z 134.518,A 54.098,B 90.000,C 0.000} C_DIS
LIN {X -170.564,Y -234.538,Z 134.568,A 53.974,B 90.000,C 0.000} C_DIS
LIN {X -171.003,Y -234.218,Z 134.833,A 53.867,B 90.000,C 0.000} C_DIS
LIN {X -171.401,Y -233.926,Z 135.340,A 53.769,B 90.000,C 0.000} C_DIS
LIN {X -172.048,Y -233.452,Z 136.635,A 53.611,B 90.000,C 0.000} C_DIS
LIN {X -172.847,Y -232.860,Z 137.832,A 53.414,B 90.000,C 0.000} C_DIS
LIN {X -172.948,Y -232.785,Z 138.120,A 53.389,B 90.000,C 0.000} C_DIS
LIN {X -172.966,Y -232.772,Z 138.399,A 53.385,B 90.000,C 0.000} C_DIS
LIN {X -172.747,Y -232.935,Z 139.003,A 53.439,B 90.000,C 0.000} C_DIS
LIN {X -171.333,Y -233.975,Z 140.784,A 53.786,B 90.000,C 0.000} C_DIS
LIN {X -169.861,Y -235.046,Z 142.496,A 54.146,B 90.000,C 0.000} C_DIS
LIN {X -168.390,Y -236.100,Z 144.221,A 54.503,B 90.000,C 0.000} C_DIS
LIN {X -166.922,Y -237.142,Z 145.956,A 54.859,B 90.000,C 0.000} C_DIS
LIN {X -165.727,Y -237.980,Z 147.390,A 55.147,B 90.000,C 0.000} C_DIS
LIN {X -165.551,Y -238.103,Z 147.762,A 55.190,B 90.000,C 0.000} C_DIS
LIN {X -165.438,Y -238.181,Z 148.292,A 55.217,B 90.000,C 0.000} C_DIS
LIN {X -165.310,Y -238.270,Z 150.787,A 55.247,B 90.000,C 0.000} C_DIS
LIN {X -165.217,Y -238.334,Z 152.684,A 55.270,B 90.000,C 0.000} C_DIS
LIN {X -164.737,Y -238.666,Z 155.115,A 55.385,B 90.000,C 0.000} C_DIS
LIN {X -164.461,Y -238.857,Z 156.155,A 55.451,B 90.000,C 0.000} C_DIS
LIN {X -164.391,Y -238.905,Z 156.802,A 55.468,B 90.000,C 0.000} C_DIS
LIN {X -164.523,Y -238.814,Z 157.403,A 55.436,B 90.000,C 0.000} C_DIS
LIN {X -164.880,Y -238.568,Z 158.047,A 55.351,B 90.000,C 0.000} C_DIS
LIN {X -165.399,Y -238.209,Z 158.647,A 55.226,B 90.000,C 0.000} C_DIS
LIN {X -166.470,Y -237.461,Z 159.418,A 54.968,B 90.000,C 0.000} C_DIS
LIN {X -166.748,Y -237.266,Z 159.728,A 54.901,B 90.000,C 0.000} C_DIS
LIN {X -166.894,Y -237.163,Z 160.115,A 54.866,B 90.000,C 0.000} C_DIS
LIN {X -166.949,Y -237.125,Z 160.647,A 54.852,B 90.000,C 0.000} C_DIS
LIN {X -166.945,Y -237.127,Z 161.122,A 54.853,B 90.000,C 0.000} C_DIS
LIN {X -166.870,Y -237.180,Z 161.477,A 54.871,B 90.000,C 0.000} C_DIS
LIN {X -166.587,Y -237.379,Z 162.050,A 54.940,B 90.000,C 0.000} C_DIS
LIN {X -166.124,Y -237.703,Z 162.465,A 55.051,B 90.000,C 0.000} C_DIS
LIN {X -165.446,Y -238.176,Z 162.741,A 55.215,B 90.000,C 0.000} C_DIS
LIN {X -164.518,Y -238.818,Z 162.898,A 55.438,B 90.000,C 0.000} C_DIS
LIN {X -163.790,Y -239.318,Z 162.908,A 55.612,B 90.000,C 0.000} C_DIS
LIN {X -163.237,Y -239.695,Z 162.522,A 55.744,B 90.000,C 0.000} C_DIS
LIN {X -162.791,Y -239.998,Z 162.068,A 55.851,B 90.000,C 0.000} C_DIS
LIN {X -162.365,Y -240.286,Z 161.456,A 55.953,B 90.000,C 0.000} C_DIS
LIN {X -161.311,Y -240.995,Z 159.303,A 56.204,B 90.000,C 0.000} C_DIS
LIN {X -160.473,Y -241.554,Z 157.535,A 56.403,B 90.000,C 0.000} C_DIS
LIN {X -159.877,Y -241.949,Z 156.572,A 56.544,B 90.000,C 0.000} C_DIS
LIN {X -159.479,Y -242.212,Z 156.289,A 56.638,B 90.000,C 0.000} C_DIS
LIN {X -158.911,Y -242.584,Z 156.217,A 56.772,B 90.000,C 0.000} C_DIS
LIN {X -158.391,Y -242.925,Z 156.276,A 56.895,B 90.000,C 0.000} C_DIS
LIN {X -157.779,Y -243.322,Z 156.502,A 57.039,B 90.000,C 0.000} C_DIS
LIN {X -155.889,Y -244.535,Z 157.600,A 57.483,B 90.000,C 0.000} C_DIS
LIN {X -154.005,Y -245.724,Z 158.735,A 57.923,B 90.000,C 0.000} C_DIS
LIN {X -152.129,Y -246.894,Z 159.901,A 58.360,B 90.000,C 0.000} C_DIS
LIN {X -151.987,Y -246.982,Z 159.992,A 58.393,B 90.000,C 0.000} C_DIS
LIN {X -151.435,Y -247.321,Z 160.505,A 58.521,B 90.000,C 0.000} C_DIS
LIN {X -151.169,Y -247.483,Z 161.067,A 58.582,B 90.000,C 0.000} C_DIS
LIN {X -151.085,Y -247.535,Z 161.814,A 58.602,B 90.000,C 0.000} C_DIS
LIN {X -151.175,Y -247.480,Z 163.018,A 58.581,B 90.000,C 0.000} C_DIS
LIN {X -151.789,Y -247.103,Z 165.412,A 58.439,B 90.000,C 0.000} C_DIS
LIN {X -152.326,Y -246.773,Z 167.831,A 58.314,B 90.000,C 0.000} C_DIS
LIN {X -152.366,Y -246.748,Z 168.044,A 58.305,B 90.000,C 0.000} C_DIS
LIN {X -152.454,Y -246.694,Z 169.619,A 58.284,B 90.000,C 0.000} C_DIS
LIN {X -152.367,Y -246.747,Z 170.974,A 58.305,B 90.000,C 0.000} C_DIS
LIN {X -152.223,Y -246.836,Z 171.485,A 58.338,B 90.000,C 0.000} C_DIS
LIN {X -151.982,Y -246.985,Z 172.016,A 58.394,B 90.000,C 0.000} C_DIS
LIN {X -150.717,Y -247.759,Z 174.028,A 58.687,B 90.000,C 0.000} C_DIS
LIN {X -150.376,Y -247.966,Z 174.600,A 58.766,B 90.000,C 0.000} C_DIS
LIN {X -150.099,Y -248.133,Z 175.246,A 58.830,B 90.000,C 0.000} C_DIS
LIN {X -149.911,Y -248.247,Z 175.968,A 58.873,B 90.000,C 0.000} C_DIS
LIN {X -149.779,Y -248.327,Z 176.863,A 58.904,B 90.000,C 0.000} C_DIS
LIN {X -149.722,Y -248.361,Z 178.741,A 58.917,B 90.000,C 0.000} C_DIS
LIN {X -149.857,Y -248.280,Z 180.641,A 58.886,B 90.000,C 0.000} C_DIS
LIN {X -150.201,Y -248.072,Z 182.247,A 58.806,B 90.000,C 0.000} C_DIS
LIN {X -150.742,Y -247.744,Z 183.763,A 58.681,B 90.000,C 0.000} C_DIS
LIN {X -151.500,Y -247.281,Z 185.238,A 58.506,B 90.000,C 0.000} C_DIS
LIN {X -152.824,Y -246.464,Z 187.195,A 58.198,B 90.000,C 0.000} C_DIS
LIN {X -154.183,Y -245.617,Z 189.114,A 57.882,B 90.000,C 0.000} C_DIS
LIN {X -154.229,Y -245.588,Z 189.177,A 57.871,B 90.000,C 0.000} C_DIS
LIN {X -154.961,Y -245.127,Z 189.672,A 57.700,B 90.000,C 0.000} C_DIS
LIN {X -155.656,Y -244.686,Z 190.026,A 57.538,B 90.000,C 0.000} C_DIS
LIN {X -156.044,Y -244.438,Z 190.021,A 57.447,B 90.000,C 0.000} C_DIS
LIN {X -156.268,Y -244.296,Z 189.766,A 57.394,B 90.000,C 0.000} C_DIS
LIN {X -156.294,Y -244.279,Z 189.393,A 57.388,B 90.000,C 0.000} C_DIS
LIN {X -155.597,Y -244.724,Z 187.837,A 57.552,B 90.000,C 0.000} C_DIS
LIN {X -155.333,Y -244.891,Z 186.818,A 57.613,B 90.000,C 0.000} C_DIS
LIN {X -155.048,Y -245.072,Z 184.341,A 57.680,B 90.000,C 0.000} C_DIS
LIN {X -155.039,Y -245.077,Z 182.874,A 57.682,B 90.000,C 0.000} C_DIS
LIN {X -155.183,Y -244.986,Z 181.711,A 57.648,B 90.000,C 0.000} C_DIS
LIN {X -155.462,Y -244.809,Z 180.784,A 57.583,B 90.000,C 0.000} C_DIS
LIN {X -155.880,Y -244.543,Z 180.084,A 57.485,B 90.000,C 0.000} C_DIS
LIN {X -156.442,Y -244.184,Z 179.600,A 57.354,B 90.000,C 0.000} C_DIS
LIN {X -157.202,Y -243.696,Z 179.273,A 57.175,B 90.000,C 0.000} C_DIS
LIN {X -158.035,Y -243.156,Z 179.167,A 56.979,B 90.000,C 0.000} C_DIS
LIN {X -158.756,Y -242.686,Z 179.230,A 56.809,B 90.000,C 0.000} C_DIS
LIN {X -159.339,Y -242.303,Z 179.466,A 56.671,B 90.000,C 0.000} C_DIS
LIN {X -159.868,Y -241.955,Z 179.908,A 56.546,B 90.000,C 0.000} C_DIS
LIN {X -160.442,Y -241.574,Z 180.630,A 56.410,B 90.000,C 0.000} C_DIS
LIN {X -160.998,Y -241.204,Z 181.540,A 56.278,B 90.000,C 0.000} C_DIS
LIN {X -161.471,Y -240.888,Z 182.544,A 56.165,B 90.000,C 0.000} C_DIS
LIN {X -162.210,Y -240.391,Z 184.880,A 55.990,B 90.000,C 0.000} C_DIS
LIN {X -162.618,Y -240.116,Z 186.194,A 55.892,B 90.000,C 0.000} C_DIS
LIN {X -163.202,Y -239.719,Z 187.582,A 55.753,B 90.000,C 0.000} C_DIS
LIN {X -164.431,Y -238.876,Z 189.589,A 55.458,B 90.000,C 0.000} C_DIS
LIN {X -165.730,Y -237.977,Z 191.527,A 55.146,B 90.000,C 0.000} C_DIS
LIN {X -166.289,Y -237.587,Z 192.388,A 55.012,B 90.000,C 0.000} C_DIS
LIN {X -166.660,Y -237.328,Z 193.160,A 54.922,B 90.000,C 0.000} C_DIS
LIN {X -166.942,Y -237.129,Z 193.947,A 54.854,B 90.000,C 0.000} C_DIS
LIN {X -167.050,Y -237.053,Z 194.395,A 54.828,B 90.000,C 0.000} C_DIS
LIN {X -167.000,Y -237.089,Z 194.661,A 54.840,B 90.000,C 0.000} C_DIS
LIN {X -166.749,Y -237.265,Z 194.800,A 54.901,B 90.000,C 0.000} C_DIS
LIN {X -165.171,Y -238.366,Z 195.107,A 55.281,B 90.000,C 0.000} C_DIS
LIN {X -164.323,Y -238.951,Z 195.562,A 55.484,B 90.000,C 0.000} C_DIS
LIN {X -163.651,Y -239.412,Z 196.305,A 55.645,B 90.000,C 0.000} C_DIS
LIN {X -163.438,Y -239.558,Z 196.689,A 55.696,B 90.000,C 0.000} C_DIS
LIN {X -163.358,Y -239.613,Z 197.004,A 55.715,B 90.000,C 0.000} C_DIS
LIN {X -163.417,Y -239.572,Z 197.274,A 55.701,B 90.000,C 0.000} C_DIS
LIN {X -163.605,Y -239.444,Z 197.579,A 55.656,B 90.000,C 0.000} C_DIS
LIN {X -165.244,Y -238.316,Z 199.093,A 55.263,B 90.000,C 0.000} C_DIS
LIN {X -166.972,Y -237.104,Z 200.432,A 54.846,B 90.000,C 0.000} C_DIS
LIN {X -168.730,Y -235.858,Z 201.699,A 54.420,B 90.000,C 0.000} C_DIS
LIN {X -170.492,Y -234.589,Z 202.939,A 53.992,B 90.000,C 0.000} C_DIS
LIN {X -172.304,Y -233.261,Z 204.035,A 53.548,B 90.000,C 0.000} C_DIS
LIN {X -174.194,Y -231.854,Z 204.869,A 53.082,B 90.000,C 0.000} C_DIS
LIN {X -175.110,Y -231.164,Z 205.165,A 52.856,B 90.000,C 0.000} C_DIS
LIN {X -175.634,Y -230.765,Z 205.163,A 52.725,B 90.000,C 0.000} C_DIS
LIN {X -175.996,Y -230.490,Z 204.953,A 52.636,B 90.000,C 0.000} C_DIS
LIN {X -176.250,Y -230.295,Z 204.587,A 52.572,B 90.000,C 0.000} C_DIS
LIN {X -176.290,Y -230.265,Z 204.456,A 52.562,B 90.000,C 0.000} C_DIS
LIN {X -176.259,Y -230.288,Z 204.317,A 52.570,B 90.000,C 0.000} C_DIS
LIN {X -175.257,Y -231.052,Z 202.815,A 52.819,B 90.000,C 0.000} C_DIS
LIN {X -174.813,Y -231.388,Z 201.937,A 52.929,B 90.000,C 0.000} C_DIS
LIN {X -174.071,Y -231.947,Z 199.616,A 53.113,B 90.000,C 0.000} C_DIS
LIN {X -173.471,Y -232.395,Z 197.231,A 53.261,B 90.000,C 0.000} C_DIS
LIN {X -173.001,Y -232.746,Z 194.801,A 53.376,B 90.000,C 0.000} C_DIS
LIN {X -172.632,Y -233.020,Z 192.343,A 53.467,B 90.000,C 0.000} C_DIS
LIN {X -172.395,Y -233.195,Z 189.861,A 53.526,B 90.000,C 0.000} C_DIS
LIN {X -172.150,Y -233.376,Z 187.379,A 53.586,B 90.000,C 0.000} C_DIS
LIN {X -171.818,Y -233.620,Z 184.914,A 53.667,B 90.000,C 0.000} C_DIS
LIN {X -171.433,Y -233.903,Z 183.195,A 53.762,B 90.000,C 0.000} C_DIS
LIN {X -170.937,Y -234.266,Z 181.756,A 53.883,B 90.000,C 0.000} C_DIS
LIN {X -170.306,Y -234.725,Z 180.356,A 54.037,B 90.000,C 0.000} C_DIS
LIN {X -169.066,Y -235.620,Z 178.379,A 54.339,B 90.000,C 0.000} C_DIS
LIN {X -168.924,Y -235.722,Z 178.180,A 54.374,B 90.000,C 0.000} C_DIS
LIN {X -168.277,Y -236.184,Z 177.466,A 54.531,B 90.000,C 0.000} C_DIS
LIN {X -166.559,Y -237.398,Z 176.116,A 54.946,B 90.000,C 0.000} C_DIS
LIN {X -164.720,Y -238.678,Z 175.006,A 55.389,B 90.000,C 0.000} C_DIS
LIN {X -164.593,Y -238.766,Z 174.939,A 55.420,B 90.000,C 0.000} C_DIS
LIN {X -162.621,Y -240.110,Z 174.192,A 55.891,B 90.000,C 0.000} C_DIS
LIN {X -160.619,Y -241.448,Z 173.521,A 56.367,B 90.000,C 0.000} C_DIS
LIN {X -158.605,Y -242.783,Z 172.878,A 56.844,B 90.000,C 0.000} C_DIS
LIN {X -157.580,Y -243.451,Z 172.548,A 57.086,B 90.000,C 0.000} C_DIS
LIN {X -157.293,Y -243.637,Z 172.069,A 57.154,B 90.000,C 0.000} C_DIS
LIN {X -156.400,Y -244.211,Z 169.806,A 57.363,B 90.000,C 0.000} C_DIS
LIN {X -155.606,Y -244.717,Z 167.490,A 57.549,B 90.000,C 0.000} C_DIS
LIN {X -155.236,Y -244.953,Z 166.194,A 57.636,B 90.000,C 0.000} C_DIS
LIN {X -155.105,Y -245.036,Z 165.254,A 57.667,B 90.000,C 0.000} C_DIS
LIN {X -155.137,Y -245.016,Z 164.448,A 57.659,B 90.000,C 0.000} C_DIS
LIN {X -155.333,Y -244.891,Z 163.764,A 57.613,B 90.000,C 0.000} C_DIS
LIN {X -155.695,Y -244.661,Z 163.188,A 57.528,B 90.000,C 0.000} C_DIS
LIN {X -156.642,Y -244.056,Z 162.384,A 57.306,B 90.000,C 0.000} C_DIS
LIN {X -157.649,Y -243.406,Z 161.731,A 57.070,B 90.000,C 0.000} C_DIS
LIN {X -157.989,Y -243.186,Z 161.717,A 56.990,B 90.000,C 0.000} C_DIS
LIN {X -158.335,Y -242.961,Z 162.091,A 56.908,B 90.000,C 0.000} C_DIS
LIN {X -158.758,Y -242.685,Z 162.846,A 56.808,B 90.000,C 0.000} C_DIS
LIN {X -159.602,Y -242.130,Z 165.133,A 56.609,B 90.000,C 0.000} C_DIS
LIN {X -160.544,Y -241.507,Z 167.362,A 56.386,B 90.000,C 0.000} C_DIS
LIN {X -160.567,Y -241.492,Z 167.412,A 56.380,B 90.000,C 0.000} C_DIS
LIN {X -161.082,Y -241.148,Z 167.793,A 56.258,B 90.000,C 0.000} C_DIS
LIN {X -161.850,Y -240.633,Z 168.129,A 56.075,B 90.000,C 0.000} C_DIS
LIN {X -162.437,Y -240.238,Z 168.240,A 55.935,B 90.000,C 0.000} C_DIS
LIN {X -164.499,Y -238.827,Z 168.330,A 55.442,B 90.000,C 0.000} C_DIS
LIN {X -166.552,Y -237.403,Z 168.392,A 54.948,B 90.000,C 0.000} C_DIS
LIN {X -167.218,Y -236.935,Z 168.394,A 54.787,B 90.000,C 0.000} C_DIS
LIN {X -167.863,Y -236.479,Z 168.277,A 54.631,B 90.000,C 0.000} C_DIS
LIN {X -168.321,Y -236.153,Z 167.987,A 54.520,B 90.000,C 0.000} C_DIS
LIN {X -168.742,Y -235.852,Z 167.469,A 54.418,B 90.000,C 0.000} C_DIS
LIN {X -169.895,Y -235.022,Z 165.413,A 54.137,B 90.000,C 0.000} C_DIS
LIN {X -170.983,Y -234.231,Z 163.306,A 53.871,B 90.000,C 0.000} C_DIS
LIN {X -171.656,Y -233.740,Z 162.003,A 53.707,B 90.000,C 0.000} C_DIS
LIN {X -172.959,Y -232.776,Z 160.099,A 53.387,B 90.000,C 0.000} C_DIS
LIN {X -173.305,Y -232.520,Z 159.586,A 53.302,B 90.000,C 0.000} C_DIS
LIN {X -173.612,Y -232.291,Z 158.613,A 53.226,B 90.000,C 0.000} C_DIS
LIN {X -173.874,Y -232.094,Z 156.324,A 53.161,B 90.000,C 0.000} C_DIS
LIN {X -173.935,Y -232.049,Z 153.825,A 53.146,B 90.000,C 0.000} C_DIS
LIN {X -173.939,Y -232.045,Z 153.649,A 53.145,B 90.000,C 0.000} C_DIS
LIN {X -173.790,Y -232.157,Z 151.156,A 53.182,B 90.000,C 0.000} C_DIS
LIN {X -173.638,Y -232.271,Z 148.664,A 53.220,B 90.000,C 0.000} C_DIS
LIN {X -173.537,Y -232.346,Z 146.167,A 53.244,B 90.000,C 0.000} C_DIS
LIN {X -173.618,Y -232.286,Z 143.669,A 53.224,B 90.000,C 0.000} C_DIS
LIN {X -173.633,Y -232.275,Z 143.476,A 53.221,B 90.000,C 0.000} C_DIS
LIN {X -173.934,Y -232.049,Z 142.840,A 53.146,B 90.000,C 0.000} C_DIS
LIN {X -175.233,Y -231.069,Z 140.943,A 52.825,B 90.000,C 0.000} C_DIS
LIN {X -176.494,Y -230.109,Z 139.009,A 52.512,B 90.000,C 0.000} C_DIS
LIN {X -176.519,Y -230.089,Z 138.967,A 52.505,B 90.000,C 0.000} C_DIS
LIN {X -176.653,Y -229.986,Z 138.485,A 52.472,B 90.000,C 0.000} C_DIS
LIN {X -176.693,Y -229.956,Z 137.980,A 52.462,B 90.000,C 0.000} C_DIS
LIN {X -176.638,Y -229.998,Z 137.467,A 52.476,B 90.000,C 0.000} C_DIS
LIN {X -176.488,Y -230.113,Z 136.957,A 52.513,B 90.000,C 0.000} C_DIS
LIN {X -176.045,Y -230.452,Z 136.228,A 52.623,B 90.000,C 0.000} C_DIS
LIN {X -174.627,Y -231.528,Z 134.473,A 52.975,B 90.000,C 0.000} C_DIS
LIN {X -174.015,Y -231.988,Z 133.698,A 53.126,B 90.000,C 0.000} C_DIS
LIN {X -173.767,Y -232.175,Z 133.225,A 53.188,B 90.000,C 0.000} C_DIS
LIN {X -173.591,Y -232.306,Z 132.418,A 53.231,B 90.000,C 0.000} C_DIS
LIN {X -173.599,Y -232.300,Z 132.043,A 53.229,B 90.000,C 0.000} C_DIS
LIN {X -173.675,Y -232.243,Z 131.731,A 53.210,B 90.000,C 0.000} C_DIS
LIN {X -173.982,Y -232.013,Z 131.281,A 53.135,B 90.000,C 0.000} C_DIS
LIN {X -174.484,Y -231.636,Z 130.921,A 53.010,B 90.000,C 0.000} C_DIS
LIN {X -175.516,Y -230.855,Z 130.345,A 52.755,B 90.000,C 0.000} C_DIS
LIN {X -175.844,Y -230.605,Z 129.979,A 52.673,B 90.000,C 0.000} C_DIS
LIN {X -176.211,Y -230.325,Z 129.414,A 52.582,B 90.000,C 0.000} C_DIS
LIN {X -176.418,Y -230.166,Z 128.859,A 52.531,B 90.000,C 0.000} C_DIS
LIN {X -176.463,Y -230.132,Z 128.321,A 52.519,B 90.000,C 0.000} C_DIS
LIN {X -176.345,Y -230.223,Z 127.810,A 52.549,B 90.000,C 0.000} C_DIS
LIN {X -176.055,Y -230.444,Z 127.340,A 52.621,B 90.000,C 0.000} C_DIS
LIN {X -174.841,Y -228.855,Z 127.340,A 52.621,B 90.000,C 0.000} C_DIS
WAIT SEC 0.1
RET=EKI_SetBool("oxy","torchState",FALSE)
RET = EKI_Send("oxy","torchState")
LIN {X -163.913,Y -214.552,Z 127.340,A 52.621,B 90.000,C 0.000} C_DIS
LIN {X -153.623,Y -222.036,Z 123.663,A 55.321,B 90.000,C 0.000} C_DIS
LIN {X -163.865,Y -236.838,Z 123.663,A 55.321,B 90.000,C 0.000} C_DIS
LIN {X -165.003,Y -238.483,Z 123.663,A 55.321,B 90.000,C 0.000} C_DIS
WAIT SEC 1
RET=EKI_SetBool("oxy","torchState",TRUE)
RET = EKI_Send("oxy","torchState")
LIN {X -165.003,Y -238.483,Z 123.663,A 55.321,B 90.000,C 0.000} C_DIS
LIN {X -163.865,Y -236.838,Z 123.663,A 55.321,B 90.000,C 0.000} C_DIS
WAIT SEC 0.1
RET=EKI_SetBool("oxy","torchState",FALSE)
RET = EKI_Send("oxy","torchState")
LIN {X -153.623,Y -222.036,Z 123.663,A 55.321,B 90.000,C 0.000} C_DIS
LIN {X -161.993,Y -216.005,Z 108.574,A 53.132,B 90.000,C 0.000} C_DIS
LIN {X -172.793,Y -230.406,Z 108.574,A 53.132,B 90.000,C 0.000} C_DIS
LIN {X -173.993,Y -232.006,Z 108.574,A 53.132,B 90.000,C 0.000} C_DIS
WAIT SEC 1
RET=EKI_SetBool("oxy","torchState",TRUE)
RET = EKI_Send("oxy","torchState")
LIN {X -174.369,Y -231.723,Z 108.751,A 53.039,B 90.000,C 0.000} C_DIS
LIN {X -174.533,Y -231.599,Z 108.789,A 52.998,B 90.000,C 0.000} C_DIS
LIN {X -175.289,Y -231.027,Z 106.475,A 52.811,B 90.000,C 0.000} C_DIS
LIN {X -176.238,Y -230.305,Z 104.278,A 52.575,B 90.000,C 0.000} C_DIS
LIN {X -177.172,Y -229.587,Z 102.305,A 52.343,B 90.000,C 0.000} C_DIS
LIN {X -178.539,Y -228.524,Z 100.502,A 52.001,B 90.000,C 0.000} C_DIS
LIN {X -179.218,Y -227.993,Z 99.682,A 51.830,B 90.000,C 0.000} C_DIS
LIN {X -179.748,Y -227.575,Z 99.197,A 51.697,B 90.000,C 0.000} C_DIS
LIN {X -179.978,Y -227.394,Z 99.082,A 51.639,B 90.000,C 0.000} C_DIS
LIN {X -180.159,Y -227.250,Z 99.116,A 51.593,B 90.000,C 0.000} C_DIS
LIN {X -181.604,Y -226.098,Z 100.311,A 51.228,B 90.000,C 0.000} C_DIS
LIN {X -183.041,Y -224.936,Z 99.113,A 50.863,B 90.000,C 0.000} C_DIS
LIN {X -183.211,Y -224.797,Z 99.074,A 50.820,B 90.000,C 0.000} C_DIS
LIN {X -183.356,Y -224.679,Z 99.137,A 50.783,B 90.000,C 0.000} C_DIS
LIN {X -184.805,Y -223.488,Z 100.791,A 50.412,B 90.000,C 0.000} C_DIS
LIN {X -186.104,Y -222.408,Z 102.525,A 50.078,B 90.000,C 0.000} C_DIS
LIN {X -187.050,Y -221.613,Z 104.699,A 49.834,B 90.000,C 0.000} C_DIS
LIN {X -187.918,Y -220.877,Z 106.924,A 49.609,B 90.000,C 0.000} C_DIS
LIN {X -188.455,Y -220.419,Z 108.649,A 49.470,B 90.000,C 0.000} C_DIS
LIN {X -188.590,Y -220.304,Z 108.741,A 49.435,B 90.000,C 0.000} C_DIS
LIN {X -188.953,Y -219.992,Z 108.614,A 49.340,B 90.000,C 0.000} C_DIS
LIN {X -189.292,Y -219.701,Z 108.241,A 49.252,B 90.000,C 0.000} C_DIS
LIN {X -190.306,Y -218.823,Z 106.132,A 48.987,B 90.000,C 0.000} C_DIS
LIN {X -191.313,Y -217.943,Z 104.020,A 48.723,B 90.000,C 0.000} C_DIS
LIN {X -191.841,Y -217.479,Z 102.949,A 48.584,B 90.000,C 0.000} C_DIS
LIN {X -192.223,Y -217.142,Z 101.948,A 48.483,B 90.000,C 0.000} C_DIS
LIN {X -192.397,Y -216.987,Z 101.038,A 48.437,B 90.000,C 0.000} C_DIS
LIN {X -192.439,Y -216.950,Z 99.968,A 48.426,B 90.000,C 0.000} C_DIS
LIN {X -192.384,Y -216.998,Z 98.855,A 48.441,B 90.000,C 0.000} C_DIS
LIN {X -192.206,Y -217.156,Z 97.980,A 48.488,B 90.000,C 0.000} C_DIS
LIN {X -191.881,Y -217.444,Z 97.268,A 48.574,B 90.000,C 0.000} C_DIS
LIN {X -191.384,Y -217.881,Z 96.646,A 48.704,B 90.000,C 0.000} C_DIS
LIN {X -190.700,Y -218.480,Z 96.053,A 48.884,B 90.000,C 0.000} C_DIS
LIN {X -189.992,Y -219.096,Z 95.643,A 49.069,B 90.000,C 0.000} C_DIS
LIN {X -189.341,Y -219.659,Z 95.461,A 49.239,B 90.000,C 0.000} C_DIS
LIN {X -188.012,Y -220.797,Z 95.519,A 49.585,B 90.000,C 0.000} C_DIS
LIN {X -187.779,Y -220.995,Z 95.416,A 49.646,B 90.000,C 0.000} C_DIS
LIN {X -187.277,Y -221.421,Z 94.872,A 49.776,B 90.000,C 0.000} C_DIS
LIN {X -186.764,Y -221.854,Z 94.060,A 49.908,B 90.000,C 0.000} C_DIS
LIN {X -185.837,Y -222.631,Z 91.872,A 50.147,B 90.000,C 0.000} C_DIS
LIN {X -185.004,Y -223.323,Z 89.955,A 50.361,B 90.000,C 0.000} C_DIS
LIN {X -184.029,Y -224.128,Z 88.222,A 50.611,B 90.000,C 0.000} C_DIS
LIN {X -183.541,Y -224.528,Z 87.561,A 50.736,B 90.000,C 0.000} C_DIS
LIN {X -183.043,Y -224.934,Z 87.022,A 50.862,B 90.000,C 0.000} C_DIS
LIN {X -182.531,Y -225.350,Z 86.598,A 50.993,B 90.000,C 0.000} C_DIS
LIN {X -181.996,Y -225.782,Z 86.277,A 51.129,B 90.000,C 0.000} C_DIS
LIN {X -181.482,Y -226.195,Z 86.219,A 51.259,B 90.000,C 0.000} C_DIS
LIN {X -180.900,Y -226.661,Z 86.437,A 51.406,B 90.000,C 0.000} C_DIS
LIN {X -180.355,Y -227.095,Z 86.837,A 51.544,B 90.000,C 0.000} C_DIS
LIN {X -179.845,Y -227.499,Z 87.327,A 51.672,B 90.000,C 0.000} C_DIS
LIN {X -179.371,Y -227.873,Z 87.910,A 51.792,B 90.000,C 0.000} C_DIS
LIN {X -178.207,Y -228.783,Z 89.927,A 52.084,B 90.000,C 0.000} C_DIS
LIN {X -177.175,Y -229.584,Z 92.058,A 52.342,B 90.000,C 0.000} C_DIS
LIN {X -176.189,Y -230.342,Z 94.227,A 52.588,B 90.000,C 0.000} C_DIS
LIN {X -176.033,Y -230.461,Z 94.569,A 52.626,B 90.000,C 0.000} C_DIS
LIN {X -175.670,Y -230.738,Z 95.084,A 52.716,B 90.000,C 0.000} C_DIS
LIN {X -175.308,Y -231.013,Z 95.389,A 52.806,B 90.000,C 0.000} C_DIS
LIN {X -174.884,Y -231.335,Z 95.523,A 52.912,B 90.000,C 0.000} C_DIS
LIN {X -173.724,Y -232.207,Z 95.428,A 53.198,B 90.000,C 0.000} C_DIS
LIN {X -173.354,Y -232.483,Z 95.488,A 53.290,B 90.000,C 0.000} C_DIS
LIN {X -172.522,Y -233.101,Z 95.831,A 53.494,B 90.000,C 0.000} C_DIS
LIN {X -171.724,Y -233.690,Z 96.387,A 53.690,B 90.000,C 0.000} C_DIS
LIN {X -171.058,Y -234.178,Z 97.074,A 53.853,B 90.000,C 0.000} C_DIS
LIN {X -170.621,Y -234.496,Z 97.810,A 53.960,B 90.000,C 0.000} C_DIS
LIN {X -170.373,Y -234.676,Z 98.680,A 54.021,B 90.000,C 0.000} C_DIS
LIN {X -170.315,Y -234.719,Z 99.854,A 54.035,B 90.000,C 0.000} C_DIS
LIN {X -170.368,Y -234.680,Z 101.009,A 54.022,B 90.000,C 0.000} C_DIS
LIN {X -170.579,Y -234.527,Z 102.011,A 53.970,B 90.000,C 0.000} C_DIS
LIN {X -171.027,Y -234.200,Z 103.112,A 53.861,B 90.000,C 0.000} C_DIS
LIN {X -172.116,Y -233.401,Z 105.215,A 53.594,B 90.000,C 0.000} C_DIS
LIN {X -173.158,Y -232.629,Z 107.353,A 53.338,B 90.000,C 0.000} C_DIS
LIN {X -173.624,Y -232.282,Z 108.169,A 53.223,B 90.000,C 0.000} C_DIS
LIN {X -173.993,Y -232.006,Z 108.574,A 53.132,B 90.000,C 0.000} C_DIS
LIN {X -172.793,Y -230.406,Z 108.574,A 53.132,B 90.000,C 0.000} C_DIS
WAIT SEC 0.1
RET=EKI_SetBool("oxy","torchState",FALSE)
RET = EKI_Send("oxy","torchState")
LIN {X -161.993,Y -216.005,Z 108.574,A 53.132,B 90.000,C 0.000} C_DIS
LIN {X -134.537,Y -234.094,Z 137.095,A 60.113,B 90.000,C 0.000} C_DIS
LIN {X -143.506,Y -249.700,Z 137.095,A 60.113,B 90.000,C 0.000} C_DIS
LIN {X -144.502,Y -251.434,Z 137.095,A 60.113,B 90.000,C 0.000} C_DIS
WAIT SEC 1
RET=EKI_SetBool("oxy","torchState",TRUE)
RET = EKI_Send("oxy","torchState")
LIN {X -144.219,Y -251.597,Z 137.025,A 60.178,B 90.000,C 0.000} C_DIS
LIN {X -143.848,Y -251.809,Z 137.363,A 60.263,B 90.000,C 0.000} C_DIS
LIN {X -143.561,Y -251.972,Z 137.764,A 60.328,B 90.000,C 0.000} C_DIS
LIN {X -143.045,Y -252.266,Z 138.807,A 60.445,B 90.000,C 0.000} C_DIS
LIN {X -142.683,Y -252.471,Z 139.275,A 60.527,B 90.000,C 0.000} C_DIS
LIN {X -142.137,Y -252.778,Z 139.835,A 60.651,B 90.000,C 0.000} C_DIS
LIN {X -141.547,Y -253.110,Z 140.283,A 60.785,B 90.000,C 0.000} C_DIS
LIN {X -139.529,Y -254.226,Z 141.250,A 61.240,B 90.000,C 0.000} C_DIS
LIN {X -137.835,Y -255.150,Z 142.040,A 61.621,B 90.000,C 0.000} C_DIS
LIN {X -137.224,Y -255.479,Z 142.465,A 61.759,B 90.000,C 0.000} C_DIS
LIN {X -136.739,Y -255.739,Z 142.940,A 61.867,B 90.000,C 0.000} C_DIS
LIN {X -136.166,Y -256.045,Z 143.870,A 61.996,B 90.000,C 0.000} C_DIS
LIN {X -135.749,Y -256.266,Z 145.148,A 62.089,B 90.000,C 0.000} C_DIS
LIN {X -135.501,Y -256.397,Z 146.614,A 62.144,B 90.000,C 0.000} C_DIS
LIN {X -135.452,Y -256.423,Z 147.953,A 62.155,B 90.000,C 0.000} C_DIS
LIN {X -135.599,Y -256.345,Z 149.096,A 62.122,B 90.000,C 0.000} C_DIS
LIN {X -135.939,Y -256.165,Z 149.976,A 62.046,B 90.000,C 0.000} C_DIS
LIN {X -136.324,Y -255.961,Z 150.430,A 61.960,B 90.000,C 0.000} C_DIS
LIN {X -136.682,Y -255.770,Z 150.662,A 61.880,B 90.000,C 0.000} C_DIS
LIN {X -137.967,Y -255.078,Z 149.113,A 61.592,B 90.000,C 0.000} C_DIS
LIN {X -138.742,Y -254.658,Z 148.358,A 61.418,B 90.000,C 0.000} C_DIS
LIN {X -140.612,Y -253.629,Z 147.056,A 60.996,B 90.000,C 0.000} C_DIS
LIN {X -142.495,Y -252.576,Z 145.793,A 60.570,B 90.000,C 0.000} C_DIS
LIN {X -142.933,Y -252.330,Z 145.490,A 60.471,B 90.000,C 0.000} C_DIS
LIN {X -144.000,Y -251.722,Z 144.493,A 60.228,B 90.000,C 0.000} C_DIS
LIN {X -144.341,Y -251.527,Z 143.863,A 60.150,B 90.000,C 0.000} C_DIS
LIN {X -144.558,Y -251.402,Z 143.193,A 60.101,B 90.000,C 0.000} C_DIS
LIN {X -144.692,Y -251.325,Z 142.394,A 60.070,B 90.000,C 0.000} C_DIS
LIN {X -144.776,Y -251.276,Z 139.895,A 60.051,B 90.000,C 0.000} C_DIS
LIN {X -144.770,Y -251.280,Z 138.104,A 60.053,B 90.000,C 0.000} C_DIS
LIN {X -144.698,Y -251.321,Z 137.508,A 60.069,B 90.000,C 0.000} C_DIS
LIN {X -144.502,Y -251.434,Z 137.095,A 60.113,B 90.000,C 0.000} C_DIS
LIN {X -143.506,Y -249.700,Z 137.095,A 60.113,B 90.000,C 0.000} C_DIS
WAIT SEC 0.1
RET=EKI_SetBool("oxy","torchState",FALSE)
RET = EKI_Send("oxy","torchState")
LIN {X -134.537,Y -234.094,Z 137.095,A 60.113,B 90.000,C 0.000} C_DIS
LIN {X -134.522,Y -234.102,Z 175.080,A 60.117,B 90.000,C 0.000} C_DIS
LIN {X -143.490,Y -249.709,Z 175.080,A 60.117,B 90.000,C 0.000} C_DIS
LIN {X -144.487,Y -251.443,Z 175.080,A 60.117,B 90.000,C 0.000} C_DIS
WAIT SEC 1
RET=EKI_SetBool("oxy","torchState",TRUE)
RET = EKI_Send("oxy","torchState")
LIN {X -144.726,Y -251.305,Z 175.238,A 60.062,B 90.000,C 0.000} C_DIS
LIN {X -145.069,Y -251.108,Z 175.871,A 59.984,B 90.000,C 0.000} C_DIS
LIN {X -145.745,Y -250.716,Z 178.245,A 59.830,B 90.000,C 0.000} C_DIS
LIN {X -146.557,Y -250.242,Z 180.562,A 59.644,B 90.000,C 0.000} C_DIS
LIN {X -147.653,Y -249.597,Z 182.714,A 59.393,B 90.000,C 0.000} C_DIS
LIN {X -148.907,Y -248.850,Z 184.744,A 59.104,B 90.000,C 0.000} C_DIS
LIN {X -150.235,Y -248.051,Z 186.705,A 58.798,B 90.000,C 0.000} C_DIS
LIN {X -151.468,Y -247.300,Z 188.413,A 58.513,B 90.000,C 0.000} C_DIS
LIN {X -153.016,Y -246.344,Z 190.128,A 58.154,B 90.000,C 0.000} C_DIS
LIN {X -154.565,Y -245.376,Z 191.835,A 57.793,B 90.000,C 0.000} C_DIS
LIN {X -155.254,Y -244.941,Z 192.616,A 57.632,B 90.000,C 0.000} C_DIS
LIN {X -155.466,Y -244.807,Z 192.979,A 57.582,B 90.000,C 0.000} C_DIS
LIN {X -155.565,Y -244.744,Z 193.376,A 57.559,B 90.000,C 0.000} C_DIS
LIN {X -155.567,Y -244.742,Z 194.453,A 57.558,B 90.000,C 0.000} C_DIS
LIN {X -155.462,Y -244.809,Z 194.820,A 57.583,B 90.000,C 0.000} C_DIS
LIN {X -155.236,Y -244.953,Z 195.254,A 57.636,B 90.000,C 0.000} C_DIS
LIN {X -154.944,Y -245.138,Z 195.591,A 57.704,B 90.000,C 0.000} C_DIS
LIN {X -154.597,Y -245.356,Z 195.821,A 57.785,B 90.000,C 0.000} C_DIS
LIN {X -154.208,Y -245.601,Z 195.933,A 57.876,B 90.000,C 0.000} C_DIS
LIN {X -153.773,Y -245.874,Z 195.898,A 57.978,B 90.000,C 0.000} C_DIS
LIN {X -153.262,Y -246.193,Z 195.691,A 58.097,B 90.000,C 0.000} C_DIS
LIN {X -151.479,Y -247.293,Z 194.328,A 58.511,B 90.000,C 0.000} C_DIS
LIN {X -151.039,Y -247.563,Z 193.955,A 58.612,B 90.000,C 0.000} C_DIS
LIN {X -150.782,Y -247.719,Z 193.825,A 58.672,B 90.000,C 0.000} C_DIS
LIN {X -150.093,Y -248.137,Z 196.192,A 58.831,B 90.000,C 0.000} C_DIS
LIN {X -149.987,Y -248.201,Z 196.491,A 58.856,B 90.000,C 0.000} C_DIS
LIN {X -149.699,Y -248.375,Z 196.981,A 58.922,B 90.000,C 0.000} C_DIS
LIN {X -149.300,Y -248.615,Z 197.433,A 59.014,B 90.000,C 0.000} C_DIS
LIN {X -148.811,Y -248.908,Z 197.828,A 59.127,B 90.000,C 0.000} C_DIS
LIN {X -148.250,Y -249.243,Z 198.148,A 59.256,B 90.000,C 0.000} C_DIS
LIN {X -146.227,Y -250.435,Z 198.684,A 59.720,B 90.000,C 0.000} C_DIS
LIN {X -145.627,Y -250.784,Z 199.046,A 59.857,B 90.000,C 0.000} C_DIS
LIN {X -144.795,Y -251.265,Z 199.940,A 60.047,B 90.000,C 0.000} C_DIS
LIN {X -144.018,Y -251.712,Z 201.028,A 60.224,B 90.000,C 0.000} C_DIS
LIN {X -143.598,Y -251.952,Z 201.828,A 60.319,B 90.000,C 0.000} C_DIS
LIN {X -142.669,Y -252.479,Z 204.088,A 60.530,B 90.000,C 0.000} C_DIS
LIN {X -142.460,Y -252.597,Z 204.590,A 60.578,B 90.000,C 0.000} C_DIS
LIN {X -142.099,Y -252.800,Z 204.401,A 60.660,B 90.000,C 0.000} C_DIS
LIN {X -141.454,Y -253.162,Z 203.833,A 60.806,B 90.000,C 0.000} C_DIS
LIN {X -140.935,Y -253.451,Z 203.063,A 60.923,B 90.000,C 0.000} C_DIS
LIN {X -140.558,Y -253.660,Z 202.001,A 61.008,B 90.000,C 0.000} C_DIS
LIN {X -140.105,Y -253.910,Z 199.555,A 61.111,B 90.000,C 0.000} C_DIS
LIN {X -139.808,Y -254.074,Z 197.079,A 61.178,B 90.000,C 0.000} C_DIS
LIN {X -139.861,Y -254.045,Z 194.580,A 61.166,B 90.000,C 0.000} C_DIS
LIN {X -139.931,Y -254.007,Z 193.978,A 61.150,B 90.000,C 0.000} C_DIS
LIN {X -140.195,Y -253.861,Z 192.838,A 61.090,B 90.000,C 0.000} C_DIS
LIN {X -141.063,Y -253.379,Z 190.544,A 60.894,B 90.000,C 0.000} C_DIS
LIN {X -142.063,Y -252.820,Z 188.322,A 60.668,B 90.000,C 0.000} C_DIS
LIN {X -142.116,Y -252.790,Z 188.206,A 60.656,B 90.000,C 0.000} C_DIS
LIN {X -143.407,Y -252.060,Z 186.194,A 60.363,B 90.000,C 0.000} C_DIS
LIN {X -143.589,Y -251.957,Z 185.925,A 60.321,B 90.000,C 0.000} C_DIS
LIN {X -143.671,Y -251.910,Z 185.488,A 60.303,B 90.000,C 0.000} C_DIS
LIN {X -143.448,Y -252.037,Z 184.932,A 60.353,B 90.000,C 0.000} C_DIS
LIN {X -143.114,Y -252.227,Z 184.292,A 60.429,B 90.000,C 0.000} C_DIS
LIN {X -142.909,Y -252.343,Z 183.631,A 60.476,B 90.000,C 0.000} C_DIS
LIN {X -142.787,Y -252.412,Z 182.756,A 60.504,B 90.000,C 0.000} C_DIS
LIN {X -142.859,Y -252.371,Z 181.987,A 60.487,B 90.000,C 0.000} C_DIS
LIN {X -143.716,Y -251.884,Z 179.833,A 60.293,B 90.000,C 0.000} C_DIS
LIN {X -143.725,Y -251.879,Z 177.333,A 60.291,B 90.000,C 0.000} C_DIS
LIN {X -143.720,Y -251.882,Z 176.997,A 60.292,B 90.000,C 0.000} C_DIS
LIN {X -143.926,Y -251.764,Z 175.715,A 60.245,B 90.000,C 0.000} C_DIS
LIN {X -144.082,Y -251.675,Z 175.321,A 60.209,B 90.000,C 0.000} C_DIS
LIN {X -144.270,Y -251.567,Z 175.109,A 60.166,B 90.000,C 0.000} C_DIS
LIN {X -144.487,Y -251.443,Z 175.080,A 60.117,B 90.000,C 0.000} C_DIS
LIN {X -143.490,Y -249.709,Z 175.080,A 60.117,B 90.000,C 0.000} C_DIS
WAIT SEC 0.1
RET=EKI_SetBool("oxy","torchState",FALSE)
RET = EKI_Send("oxy","torchState")
LIN {X -134.522,Y -234.102,Z 175.080,A 60.117,B 90.000,C 0.000} C_DIS
LIN {X -145.725,Y -227.298,Z 181.639,A 57.335,B 90.000,C 0.000} C_DIS
LIN {X -155.440,Y -242.451,Z 181.639,A 57.335,B 90.000,C 0.000} C_DIS
LIN {X -156.520,Y -244.134,Z 181.639,A 57.335,B 90.000,C 0.000} C_DIS
WAIT SEC 1
RET=EKI_SetBool("oxy","torchState",TRUE)
RET = EKI_Send("oxy","torchState")
LIN {X -156.240,Y -244.313,Z 182.585,A 57.401,B 90.000,C 0.000} C_DIS
LIN {X -156.170,Y -244.358,Z 183.719,A 57.417,B 90.000,C 0.000} C_DIS
LIN {X -156.211,Y -244.332,Z 184.649,A 57.408,B 90.000,C 0.000} C_DIS
LIN {X -156.354,Y -244.241,Z 185.630,A 57.374,B 90.000,C 0.000} C_DIS
LIN {X -156.979,Y -243.839,Z 188.017,A 57.227,B 90.000,C 0.000} C_DIS
LIN {X -157.396,Y -243.570,Z 189.693,A 57.129,B 90.000,C 0.000} C_DIS
LIN {X -156.933,Y -243.869,Z 191.728,A 57.238,B 90.000,C 0.000} C_DIS
LIN {X -156.732,Y -243.998,Z 193.135,A 57.285,B 90.000,C 0.000} C_DIS
LIN {X -156.648,Y -244.052,Z 195.633,A 57.305,B 90.000,C 0.000} C_DIS
LIN {X -156.717,Y -244.008,Z 198.131,A 57.289,B 90.000,C 0.000} C_DIS
LIN {X -156.727,Y -244.001,Z 198.443,A 57.287,B 90.000,C 0.000} C_DIS
LIN {X -157.201,Y -243.696,Z 200.878,A 57.175,B 90.000,C 0.000} C_DIS
LIN {X -157.855,Y -243.273,Z 203.253,A 57.021,B 90.000,C 0.000} C_DIS
LIN {X -157.871,Y -243.263,Z 203.300,A 57.017,B 90.000,C 0.000} C_DIS
LIN {X -158.068,Y -243.134,Z 203.599,A 56.971,B 90.000,C 0.000} C_DIS
LIN {X -158.313,Y -242.975,Z 203.763,A 56.913,B 90.000,C 0.000} C_DIS
LIN {X -158.599,Y -242.789,Z 203.790,A 56.846,B 90.000,C 0.000} C_DIS
LIN {X -158.919,Y -242.580,Z 203.677,A 56.770,B 90.000,C 0.000} C_DIS
LIN {X -159.294,Y -242.333,Z 203.391,A 56.682,B 90.000,C 0.000} C_DIS
LIN {X -159.616,Y -242.122,Z 202.942,A 56.606,B 90.000,C 0.000} C_DIS
LIN {X -159.919,Y -241.921,Z 202.267,A 56.534,B 90.000,C 0.000} C_DIS
LIN {X -160.718,Y -241.391,Z 199.958,A 56.344,B 90.000,C 0.000} C_DIS
LIN {X -161.644,Y -240.772,Z 197.720,A 56.124,B 90.000,C 0.000} C_DIS
LIN {X -162.551,Y -240.161,Z 195.472,A 55.908,B 90.000,C 0.000} C_DIS
LIN {X -162.704,Y -240.057,Z 195.141,A 55.872,B 90.000,C 0.000} C_DIS
LIN {X -163.111,Y -239.781,Z 194.502,A 55.774,B 90.000,C 0.000} C_DIS
LIN {X -164.383,Y -238.910,Z 193.047,A 55.470,B 90.000,C 0.000} C_DIS
LIN {X -164.535,Y -238.806,Z 192.725,A 55.433,B 90.000,C 0.000} C_DIS
LIN {X -164.578,Y -238.776,Z 192.411,A 55.423,B 90.000,C 0.000} C_DIS
LIN {X -164.548,Y -238.797,Z 192.208,A 55.430,B 90.000,C 0.000} C_DIS
LIN {X -164.420,Y -238.885,Z 191.956,A 55.461,B 90.000,C 0.000} C_DIS
LIN {X -163.010,Y -239.848,Z 190.130,A 55.798,B 90.000,C 0.000} C_DIS
LIN {X -162.605,Y -240.124,Z 189.603,A 55.895,B 90.000,C 0.000} C_DIS
LIN {X -161.825,Y -240.650,Z 188.327,A 56.081,B 90.000,C 0.000} C_DIS
LIN {X -160.869,Y -241.291,Z 186.273,A 56.309,B 90.000,C 0.000} C_DIS
LIN {X -160.101,Y -241.800,Z 183.949,A 56.491,B 90.000,C 0.000} C_DIS
LIN {X -159.322,Y -242.315,Z 181.630,A 56.675,B 90.000,C 0.000} C_DIS
LIN {X -159.217,Y -242.384,Z 181.363,A 56.700,B 90.000,C 0.000} C_DIS
LIN {X -158.879,Y -242.606,Z 180.810,A 56.780,B 90.000,C 0.000} C_DIS
LIN {X -158.507,Y -242.849,Z 180.493,A 56.868,B 90.000,C 0.000} C_DIS
LIN {X -158.246,Y -243.019,Z 180.386,A 56.929,B 90.000,C 0.000} C_DIS
LIN {X -157.911,Y -243.237,Z 180.375,A 57.008,B 90.000,C 0.000} C_DIS
LIN {X -157.470,Y -243.523,Z 180.465,A 57.112,B 90.000,C 0.000} C_DIS
LIN {X -157.101,Y -243.760,Z 180.696,A 57.199,B 90.000,C 0.000} C_DIS
LIN {X -156.790,Y -243.961,Z 181.083,A 57.272,B 90.000,C 0.000} C_DIS
LIN {X -156.520,Y -244.134,Z 181.639,A 57.335,B 90.000,C 0.000} C_DIS
LIN {X -155.440,Y -242.451,Z 181.639,A 57.335,B 90.000,C 0.000} C_DIS
WAIT SEC 0.1
RET=EKI_SetBool("oxy","torchState",FALSE)
RET = EKI_Send("oxy","torchState")
LIN {X -145.725,Y -227.298,Z 181.639,A 57.335,B 90.000,C 0.000} C_DIS
LIN {X -152.098,Y -223.083,Z 200.854,A 55.714,B 90.000,C 0.000} C_DIS
LIN {X -162.238,Y -237.955,Z 200.854,A 55.714,B 90.000,C 0.000} C_DIS
LIN {X -163.365,Y -239.608,Z 200.854,A 55.714,B 90.000,C 0.000} C_DIS
WAIT SEC 1
RET=EKI_SetBool("oxy","torchState",TRUE)
RET = EKI_Send("oxy","torchState")
LIN {X -162.778,Y -240.007,Z 200.842,A 55.854,B 90.000,C 0.000} C_DIS
LIN {X -162.424,Y -240.246,Z 201.042,A 55.938,B 90.000,C 0.000} C_DIS
LIN {X -162.275,Y -240.347,Z 201.343,A 55.974,B 90.000,C 0.000} C_DIS
LIN {X -162.413,Y -240.254,Z 201.753,A 55.941,B 90.000,C 0.000} C_DIS
LIN {X -162.752,Y -240.024,Z 202.236,A 55.860,B 90.000,C 0.000} C_DIS
LIN {X -163.340,Y -239.625,Z 202.796,A 55.720,B 90.000,C 0.000} C_DIS
LIN {X -165.146,Y -238.383,Z 203.998,A 55.287,B 90.000,C 0.000} C_DIS
LIN {X -166.930,Y -237.137,Z 205.230,A 54.857,B 90.000,C 0.000} C_DIS
LIN {X -168.621,Y -235.938,Z 206.348,A 54.447,B 90.000,C 0.000} C_DIS
LIN {X -170.510,Y -234.577,Z 207.258,A 53.987,B 90.000,C 0.000} C_DIS
LIN {X -172.397,Y -233.189,Z 208.130,A 53.524,B 90.000,C 0.000} C_DIS
LIN {X -174.298,Y -231.768,Z 208.915,A 53.055,B 90.000,C 0.000} C_DIS
LIN {X -176.206,Y -230.325,Z 209.642,A 52.583,B 90.000,C 0.000} C_DIS
LIN {X -177.378,Y -229.428,Z 210.078,A 52.291,B 90.000,C 0.000} C_DIS
LIN {X -177.600,Y -229.255,Z 212.562,A 52.236,B 90.000,C 0.000} C_DIS
LIN {X -177.860,Y -229.054,Z 215.040,A 52.171,B 90.000,C 0.000} C_DIS
LIN {X -178.236,Y -228.761,Z 217.494,A 52.077,B 90.000,C 0.000} C_DIS
LIN {X -178.797,Y -228.324,Z 219.891,A 51.936,B 90.000,C 0.000} C_DIS
LIN {X -178.835,Y -228.294,Z 220.035,A 51.926,B 90.000,C 0.000} C_DIS
LIN {X -179.337,Y -227.900,Z 221.337,A 51.800,B 90.000,C 0.000} C_DIS
LIN {X -179.935,Y -227.428,Z 222.417,A 51.650,B 90.000,C 0.000} C_DIS
LIN {X -180.557,Y -226.934,Z 223.166,A 51.493,B 90.000,C 0.000} C_DIS
LIN {X -180.855,Y -226.697,Z 223.383,A 51.418,B 90.000,C 0.000} C_DIS
LIN {X -181.131,Y -226.476,Z 223.477,A 51.348,B 90.000,C 0.000} C_DIS
LIN {X -181.334,Y -226.314,Z 223.480,A 51.297,B 90.000,C 0.000} C_DIS
LIN {X -181.382,Y -226.276,Z 223.396,A 51.284,B 90.000,C 0.000} C_DIS
LIN {X -181.436,Y -226.232,Z 220.897,A 51.271,B 90.000,C 0.000} C_DIS
LIN {X -181.475,Y -226.201,Z 219.952,A 51.261,B 90.000,C 0.000} C_DIS
LIN {X -181.735,Y -225.992,Z 218.305,A 51.195,B 90.000,C 0.000} C_DIS
LIN {X -182.230,Y -225.593,Z 216.689,A 51.069,B 90.000,C 0.000} C_DIS
LIN {X -183.174,Y -224.827,Z 214.504,A 50.829,B 90.000,C 0.000} C_DIS
LIN {X -184.142,Y -224.035,Z 212.340,A 50.582,B 90.000,C 0.000} C_DIS
LIN {X -184.243,Y -223.952,Z 212.113,A 50.556,B 90.000,C 0.000} C_DIS
LIN {X -184.758,Y -223.527,Z 210.546,A 50.424,B 90.000,C 0.000} C_DIS
LIN {X -184.824,Y -223.473,Z 210.402,A 50.407,B 90.000,C 0.000} C_DIS
LIN {X -184.950,Y -223.369,Z 210.324,A 50.375,B 90.000,C 0.000} C_DIS
LIN {X -186.805,Y -221.820,Z 209.683,A 49.898,B 90.000,C 0.000} C_DIS
LIN {X -187.693,Y -221.069,Z 209.442,A 49.668,B 90.000,C 0.000} C_DIS
LIN {X -189.479,Y -219.539,Z 208.594,A 49.203,B 90.000,C 0.000} C_DIS
LIN {X -191.261,Y -217.985,Z 207.782,A 48.736,B 90.000,C 0.000} C_DIS
LIN {X -192.996,Y -216.450,Z 206.842,A 48.278,B 90.000,C 0.000} C_DIS
LIN {X -194.690,Y -214.930,Z 205.808,A 47.829,B 90.000,C 0.000} C_DIS
LIN {X -196.323,Y -213.441,Z 204.639,A 47.392,B 90.000,C 0.000} C_DIS
LIN {X -197.903,Y -211.977,Z 203.371,A 46.967,B 90.000,C 0.000} C_DIS
LIN {X -198.671,Y -211.258,Z 202.838,A 46.759,B 90.000,C 0.000} C_DIS
LIN {X -199.157,Y -210.800,Z 202.343,A 46.627,B 90.000,C 0.000} C_DIS
LIN {X -199.500,Y -210.475,Z 201.829,A 46.533,B 90.000,C 0.000} C_DIS
LIN {X -199.631,Y -210.351,Z 201.383,A 46.498,B 90.000,C 0.000} C_DIS
LIN {X -199.561,Y -210.418,Z 201.081,A 46.517,B 90.000,C 0.000} C_DIS
LIN {X -199.367,Y -210.601,Z 200.866,A 46.570,B 90.000,C 0.000} C_DIS
LIN {X -199.367,Y -210.601,Z 200.866,A 46.570,B 90.000,C 0.000} C_DIS
LIN {X -199.129,Y -210.827,Z 200.801,A 46.634,B 90.000,C 0.000} C_DIS
LIN {X -198.796,Y -211.140,Z 200.855,A 46.725,B 90.000,C 0.000} C_DIS
LIN {X -197.082,Y -212.738,Z 201.727,A 47.188,B 90.000,C 0.000} C_DIS
LIN {X -195.374,Y -214.308,Z 202.656,A 47.646,B 90.000,C 0.000} C_DIS
LIN {X -193.634,Y -215.883,Z 203.518,A 48.110,B 90.000,C 0.000} C_DIS
LIN {X -191.872,Y -217.450,Z 204.349,A 48.576,B 90.000,C 0.000} C_DIS
LIN {X -190.080,Y -219.018,Z 205.110,A 49.046,B 90.000,C 0.000} C_DIS
LIN {X -188.254,Y -220.589,Z 205.779,A 49.522,B 90.000,C 0.000} C_DIS
LIN {X -186.395,Y -222.161,Z 206.348,A 50.003,B 90.000,C 0.000} C_DIS
LIN {X -184.517,Y -223.724,Z 206.876,A 50.486,B 90.000,C 0.000} C_DIS
LIN {X -182.673,Y -225.234,Z 207.349,A 50.957,B 90.000,C 0.000} C_DIS
LIN {X -180.725,Y -226.800,Z 207.349,A 51.451,B 90.000,C 0.000} C_DIS
LIN {X -180.618,Y -226.886,Z 207.342,A 51.478,B 90.000,C 0.000} C_DIS
LIN {X -178.690,Y -228.397,Z 206.844,A 51.962,B 90.000,C 0.000} C_DIS
LIN {X -176.761,Y -229.901,Z 206.328,A 52.445,B 90.000,C 0.000} C_DIS
LIN {X -174.829,Y -231.375,Z 205.741,A 52.925,B 90.000,C 0.000} C_DIS
LIN {X -172.894,Y -232.824,Z 205.104,A 53.403,B 90.000,C 0.000} C_DIS
LIN {X -170.969,Y -234.241,Z 204.372,A 53.875,B 90.000,C 0.000} C_DIS
LIN {X -169.043,Y -235.634,Z 203.595,A 54.344,B 90.000,C 0.000} C_DIS
LIN {X -167.148,Y -236.983,Z 202.680,A 54.804,B 90.000,C 0.000} C_DIS
LIN {X -165.246,Y -238.312,Z 201.752,A 55.263,B 90.000,C 0.000} C_DIS
LIN {X -163.365,Y -239.608,Z 200.854,A 55.714,B 90.000,C 0.000} C_DIS
LIN {X -162.238,Y -237.955,Z 200.854,A 55.714,B 90.000,C 0.000} C_DIS
WAIT SEC 0.1
RET=EKI_SetBool("oxy","torchState",FALSE)
RET = EKI_Send("oxy","torchState")
LIN {X -152.098,Y -223.083,Z 200.854,A 55.714,B 90.000,C 0.000} C_DIS
LIN {X -184.029,Y -197.569,Z 192.742,A 47.032,B 90.000,C 0.000} C_DIS
LIN {X -196.297,Y -210.740,Z 192.742,A 47.032,B 90.000,C 0.000} C_DIS
LIN {X -197.661,Y -212.203,Z 192.742,A 47.032,B 90.000,C 0.000} C_DIS
WAIT SEC 1
RET=EKI_SetBool("oxy","torchState",TRUE)
RET = EKI_Send("oxy","torchState")
LIN {X -197.866,Y -212.012,Z 193.205,A 46.977,B 90.000,C 0.000} C_DIS
LIN {X -198.861,Y -211.079,Z 194.411,A 46.707,B 90.000,C 0.000} C_DIS
LIN {X -199.252,Y -210.710,Z 195.068,A 46.601,B 90.000,C 0.000} C_DIS
LIN {X -200.076,Y -209.927,Z 197.294,A 46.376,B 90.000,C 0.000} C_DIS
LIN {X -200.857,Y -209.181,Z 199.549,A 46.163,B 90.000,C 0.000} C_DIS
LIN {X -201.625,Y -208.440,Z 201.810,A 45.952,B 90.000,C 0.000} C_DIS
LIN {X -202.032,Y -208.046,Z 203.040,A 45.840,B 90.000,C 0.000} C_DIS
LIN {X -202.207,Y -207.876,Z 203.364,A 45.792,B 90.000,C 0.000} C_DIS
LIN {X -202.415,Y -207.673,Z 203.590,A 45.735,B 90.000,C 0.000} C_DIS
LIN {X -202.652,Y -207.442,Z 203.714,A 45.669,B 90.000,C 0.000} C_DIS
LIN {X -202.911,Y -207.189,Z 203.733,A 45.598,B 90.000,C 0.000} C_DIS
LIN {X -203.199,Y -206.906,Z 203.593,A 45.518,B 90.000,C 0.000} C_DIS
LIN {X -203.445,Y -206.665,Z 203.216,A 45.450,B 90.000,C 0.000} C_DIS
LIN {X -203.676,Y -206.436,Z 202.539,A 45.386,B 90.000,C 0.000} C_DIS
LIN {X -204.177,Y -205.941,Z 200.141,A 45.246,B 90.000,C 0.000} C_DIS
LIN {X -204.349,Y -205.770,Z 198.885,A 45.199,B 90.000,C 0.000} C_DIS
LIN {X -204.496,Y -205.624,Z 196.394,A 45.158,B 90.000,C 0.000} C_DIS
LIN {X -204.474,Y -205.646,Z 193.894,A 45.164,B 90.000,C 0.000} C_DIS
LIN {X -204.240,Y -205.879,Z 191.416,A 45.229,B 90.000,C 0.000} C_DIS
LIN {X -204.220,Y -205.898,Z 191.265,A 45.234,B 90.000,C 0.000} C_DIS
LIN {X -203.874,Y -206.241,Z 189.804,A 45.331,B 90.000,C 0.000} C_DIS
LIN {X -203.856,Y -206.259,Z 189.463,A 45.336,B 90.000,C 0.000} C_DIS
LIN {X -204.445,Y -205.675,Z 187.105,A 45.172,B 90.000,C 0.000} C_DIS
LIN {X -204.635,Y -205.486,Z 186.366,A 45.119,B 90.000,C 0.000} C_DIS
LIN {X -204.895,Y -205.227,Z 184.554,A 45.046,B 90.000,C 0.000} C_DIS
LIN {X -204.921,Y -205.201,Z 183.743,A 45.039,B 90.000,C 0.000} C_DIS
LIN {X -204.878,Y -205.243,Z 182.989,A 45.051,B 90.000,C 0.000} C_DIS
LIN {X -204.767,Y -205.354,Z 182.289,A 45.082,B 90.000,C 0.000} C_DIS
LIN {X -204.588,Y -205.533,Z 181.639,A 45.132,B 90.000,C 0.000} C_DIS
LIN {X -204.238,Y -205.880,Z 180.909,A 45.229,B 90.000,C 0.000} C_DIS
LIN {X -203.820,Y -206.294,Z 180.439,A 45.346,B 90.000,C 0.000} C_DIS
LIN {X -203.404,Y -206.705,Z 180.307,A 45.461,B 90.000,C 0.000} C_DIS
LIN {X -202.969,Y -207.132,Z 180.467,A 45.582,B 90.000,C 0.000} C_DIS
LIN {X -202.639,Y -207.454,Z 180.764,A 45.673,B 90.000,C 0.000} C_DIS
LIN {X -202.360,Y -207.727,Z 181.265,A 45.750,B 90.000,C 0.000} C_DIS
LIN {X -201.664,Y -208.403,Z 183.568,A 45.942,B 90.000,C 0.000} C_DIS
LIN {X -200.996,Y -209.047,Z 185.890,A 46.125,B 90.000,C 0.000} C_DIS
LIN {X -200.276,Y -209.737,Z 187.866,A 46.322,B 90.000,C 0.000} C_DIS
LIN {X -199.482,Y -210.492,Z 189.432,A 46.538,B 90.000,C 0.000} C_DIS
LIN {X -198.256,Y -211.647,Z 191.278,A 46.871,B 90.000,C 0.000} C_DIS
LIN {X -197.694,Y -212.172,Z 192.119,A 47.023,B 90.000,C 0.000} C_DIS
LIN {X -197.618,Y -212.243,Z 192.424,A 47.044,B 90.000,C 0.000} C_DIS
LIN {X -197.661,Y -212.203,Z 192.742,A 47.032,B 90.000,C 0.000} C_DIS
LIN {X -196.297,Y -210.740,Z 192.742,A 47.032,B 90.000,C 0.000} C_DIS
WAIT SEC 0.1
RET=EKI_SetBool("oxy","torchState",FALSE)
RET = EKI_Send("oxy","torchState")
LIN {X -184.029,Y -197.569,Z 192.742,A 47.032,B 90.000,C 0.000} C_DIS
LIN {X -185.618,Y -196.076,Z 200.866,A 46.570,B 90.000,C 0.000} C_DIS
LIN {X -197.992,Y -209.148,Z 200.866,A 46.570,B 90.000,C 0.000} C_DIS
LIN {X -199.367,Y -210.601,Z 200.866,A 46.570,B 90.000,C 0.000} C_DIS
WAIT SEC 1
RET=EKI_SetBool("oxy","torchState",TRUE)
RET = EKI_Send("oxy","torchState")
LIN {X -199.367,Y -210.601,Z 200.866,A 46.570,B 90.000,C 0.000} C_DIS
LIN {X -197.992,Y -209.148,Z 200.866,A 46.570,B 90.000,C 0.000} C_DIS
WAIT SEC 0.1
RET=EKI_SetBool("oxy","torchState",FALSE)
RET = EKI_Send("oxy","torchState")
LIN {X -185.618,Y -196.077,Z 200.866,A 46.570,B 90.000,C 0.000} C_DIS
LIN {X -191.525,Y -190.311,Z 195.329,A 44.818,B 90.000,C 0.000} C_DIS
LIN {X -204.293,Y -202.998,Z 195.329,A 44.818,B 90.000,C 0.000} C_DIS
LIN {X -205.712,Y -204.408,Z 195.329,A 44.818,B 90.000,C 0.000} C_DIS
WAIT SEC 1
RET=EKI_SetBool("oxy","torchState",TRUE)
RET = EKI_Send("oxy","torchState")
LIN {X -205.469,Y -204.652,Z 194.682,A 44.886,B 90.000,C 0.000} C_DIS
LIN {X -205.388,Y -204.733,Z 193.929,A 44.909,B 90.000,C 0.000} C_DIS
LIN {X -205.490,Y -204.631,Z 193.160,A 44.880,B 90.000,C 0.000} C_DIS
LIN {X -205.736,Y -204.383,Z 192.551,A 44.811,B 90.000,C 0.000} C_DIS
LIN {X -207.002,Y -203.098,Z 190.821,A 44.454,B 90.000,C 0.000} C_DIS
LIN {X -208.242,Y -201.827,Z 189.060,A 44.104,B 90.000,C 0.000} C_DIS
LIN {X -209.435,Y -200.590,Z 187.245,A 43.764,B 90.000,C 0.000} C_DIS
LIN {X -210.541,Y -199.428,Z 185.327,A 43.447,B 90.000,C 0.000} C_DIS
LIN {X -211.560,Y -198.348,Z 183.316,A 43.154,B 90.000,C 0.000} C_DIS
LIN {X -212.452,Y -197.393,Z 181.185,A 42.896,B 90.000,C 0.000} C_DIS
LIN {X -213.175,Y -196.612,Z 178.923,A 42.685,B 90.000,C 0.000} C_DIS
LIN {X -213.719,Y -196.021,Z 176.556,A 42.527,B 90.000,C 0.000} C_DIS
LIN {X -213.851,Y -195.877,Z 175.971,A 42.488,B 90.000,C 0.000} C_DIS
LIN {X -214.083,Y -195.623,Z 175.321,A 42.420,B 90.000,C 0.000} C_DIS
LIN {X -214.317,Y -195.367,Z 175.065,A 42.352,B 90.000,C 0.000} C_DIS
LIN {X -214.561,Y -195.098,Z 175.182,A 42.280,B 90.000,C 0.000} C_DIS
LIN {X -214.736,Y -194.907,Z 175.577,A 42.229,B 90.000,C 0.000} C_DIS
LIN {X -214.878,Y -194.749,Z 176.293,A 42.187,B 90.000,C 0.000} C_DIS
LIN {X -214.927,Y -194.696,Z 176.927,A 42.172,B 90.000,C 0.000} C_DIS
LIN {X -214.935,Y -194.687,Z 179.427,A 42.170,B 90.000,C 0.000} C_DIS
LIN {X -214.940,Y -194.681,Z 179.792,A 42.169,B 90.000,C 0.000} C_DIS
LIN {X -215.056,Y -194.554,Z 180.300,A 42.135,B 90.000,C 0.000} C_DIS
LIN {X -215.593,Y -193.958,Z 182.043,A 41.976,B 90.000,C 0.000} C_DIS
LIN {X -215.646,Y -193.899,Z 182.925,A 41.960,B 90.000,C 0.000} C_DIS
LIN {X -215.511,Y -194.049,Z 183.882,A 42.000,B 90.000,C 0.000} C_DIS
LIN {X -214.950,Y -194.670,Z 185.486,A 42.166,B 90.000,C 0.000} C_DIS
LIN {X -215.015,Y -194.599,Z 185.842,A 42.147,B 90.000,C 0.000} C_DIS
LIN {X -215.956,Y -193.552,Z 187.908,A 41.869,B 90.000,C 0.000} C_DIS
LIN {X -216.792,Y -192.616,Z 190.070,A 41.620,B 90.000,C 0.000} C_DIS
LIN {X -217.501,Y -191.816,Z 192.330,A 41.409,B 90.000,C 0.000} C_DIS
LIN {X -217.571,Y -191.737,Z 192.566,A 41.388,B 90.000,C 0.000} C_DIS
LIN {X -217.829,Y -191.443,Z 193.815,A 41.311,B 90.000,C 0.000} C_DIS
LIN {X -217.969,Y -191.284,Z 195.001,A 41.269,B 90.000,C 0.000} C_DIS
LIN {X -217.995,Y -191.255,Z 196.173,A 41.262,B 90.000,C 0.000} C_DIS
LIN {X -217.786,Y -191.492,Z 198.653,A 41.324,B 90.000,C 0.000} C_DIS
LIN {X -217.517,Y -191.798,Z 201.119,A 41.405,B 90.000,C 0.000} C_DIS
LIN {X -217.498,Y -191.819,Z 201.286,A 41.410,B 90.000,C 0.000} C_DIS
LIN {X -217.166,Y -192.195,Z 202.892,A 41.509,B 90.000,C 0.000} C_DIS
LIN {X -216.789,Y -192.620,Z 203.650,A 41.621,B 90.000,C 0.000} C_DIS
LIN {X -216.218,Y -193.261,Z 204.340,A 41.791,B 90.000,C 0.000} C_DIS
LIN {X -215.957,Y -193.553,Z 204.560,A 41.869,B 90.000,C 0.000} C_DIS
LIN {X -215.869,Y -193.650,Z 204.507,A 41.894,B 90.000,C 0.000} C_DIS
LIN {X -215.141,Y -194.459,Z 202.256,A 42.109,B 90.000,C 0.000} C_DIS
LIN {X -214.810,Y -194.824,Z 201.280,A 42.207,B 90.000,C 0.000} C_DIS
LIN {X -214.501,Y -195.165,Z 200.665,A 42.298,B 90.000,C 0.000} C_DIS
LIN {X -213.407,Y -196.360,Z 199.011,A 42.618,B 90.000,C 0.000} C_DIS
LIN {X -213.016,Y -196.784,Z 198.718,A 42.732,B 90.000,C 0.000} C_DIS
LIN {X -211.370,Y -198.551,Z 198.153,A 43.209,B 90.000,C 0.000} C_DIS
LIN {X -210.794,Y -199.163,Z 197.727,A 43.375,B 90.000,C 0.000} C_DIS
LIN {X -210.430,Y -199.548,Z 197.263,A 43.480,B 90.000,C 0.000} C_DIS
LIN {X -210.111,Y -199.883,Z 196.725,A 43.571,B 90.000,C 0.000} C_DIS
LIN {X -209.712,Y -200.302,Z 195.557,A 43.685,B 90.000,C 0.000} C_DIS
LIN {X -209.422,Y -200.605,Z 194.143,A 43.768,B 90.000,C 0.000} C_DIS
LIN {X -209.322,Y -200.709,Z 193.814,A 43.797,B 90.000,C 0.000} C_DIS
LIN {X -207.885,Y -202.197,Z 195.218,A 44.205,B 90.000,C 0.000} C_DIS
LIN {X -207.484,Y -202.609,Z 195.595,A 44.319,B 90.000,C 0.000} C_DIS
LIN {X -206.961,Y -203.143,Z 195.922,A 44.467,B 90.000,C 0.000} C_DIS
LIN {X -206.517,Y -203.594,Z 195.976,A 44.592,B 90.000,C 0.000} C_DIS
LIN {X -206.095,Y -204.021,Z 195.781,A 44.710,B 90.000,C 0.000} C_DIS
LIN {X -205.712,Y -204.408,Z 195.329,A 44.818,B 90.000,C 0.000} C_DIS
LIN {X -204.293,Y -202.998,Z 195.329,A 44.818,B 90.000,C 0.000} C_DIS
WAIT SEC 0.1
RET=EKI_SetBool("oxy","torchState",FALSE)
RET = EKI_Send("oxy","torchState")
LIN {X -191.525,Y -190.311,Z 195.329,A 44.818,B 90.000,C 0.000} C_DIS
LIN {X -173.027,Y -207.272,Z 55.797,A 50.146,B 90.000,C 0.000} C_DIS
LIN {X -184.562,Y -221.090,Z 55.797,A 50.146,B 90.000,C 0.000} C_DIS
LIN {X -185.844,Y -222.626,Z 55.797,A 50.146,B 90.000,C 0.000} C_DIS
WAIT SEC 1
RET=EKI_SetBool("oxy","torchState",TRUE)
RET = EKI_Send("oxy","torchState")
LIN {X -185.844,Y -222.626,Z 55.797,A 50.146,B 90.000,C 0.000} C_DIS
LIN {X -184.562,Y -221.090,Z 55.797,A 50.146,B 90.000,C 0.000} C_DIS
WAIT SEC 0.1
RET=EKI_SetBool("oxy","torchState",FALSE)
RET = EKI_Send("oxy","torchState")
LIN {X -173.027,Y -207.272,Z 55.797,A 50.146,B 90.000,C 0.000} C_DIS
LIN {X -2.679,Y -269.987,Z 84.495,A 89.431,B 90.000,C 0.000} C_DIS
LIN {X -2.858,Y -287.986,Z 84.495,A 89.431,B 90.000,C 0.000} C_DIS
LIN {X -2.878,Y -289.986,Z 84.495,A 89.431,B 90.000,C 0.000} C_DIS
WAIT SEC 1
RET=EKI_SetBool("oxy","torchState",TRUE)
RET = EKI_Send("oxy","torchState")
LIN {X -2.310,Y -289.991,Z 83.414,A 89.544,B 90.000,C 0.000} C_DIS
LIN {X -2.226,Y -289.991,Z 83.299,A 89.560,B 90.000,C 0.000} C_DIS
LIN {X -2.084,Y -289.993,Z 83.174,A 89.588,B 90.000,C 0.000} C_DIS
LIN {X -1.970,Y -289.993,Z 83.000,A 89.611,B 90.000,C 0.000} C_DIS
LIN {X -1.193,Y -289.998,Z 82.503,A 89.764,B 90.000,C 0.000} C_DIS
LIN {X -1.116,Y -289.998,Z 82.418,A 89.779,B 90.000,C 0.000} C_DIS
LIN {X -1.070,Y -289.998,Z 82.333,A 89.789,B 90.000,C 0.000} C_DIS
LIN {X -0.403,Y -290.000,Z 81.919,A 89.920,B 90.000,C 0.000} C_DIS
LIN {X -0.205,Y -290.000,Z 81.889,A 89.959,B 90.000,C 0.000} C_DIS
LIN {X -0.129,Y -290.000,Z 81.998,A 89.974,B 90.000,C 0.000} C_DIS
LIN {X -0.383,Y -290.000,Z 83.570,A 89.924,B 90.000,C 0.000} C_DIS
LIN {X -0.261,Y -290.000,Z 84.779,A 89.948,B 90.000,C 0.000} C_DIS
LIN {X -0.223,Y -290.000,Z 84.893,A 89.956,B 90.000,C 0.000} C_DIS
LIN {X -0.210,Y -290.000,Z 85.007,A 89.959,B 90.000,C 0.000} C_DIS
LIN {X 0.224,Y -290.000,Z 86.083,A 90.044,B 90.000,C 0.000} C_DIS
LIN {X 0.235,Y -290.000,Z 86.154,A 90.046,B 90.000,C 0.000} C_DIS
LIN {X 1.684,Y -289.995,Z 88.191,A 90.333,B 90.000,C 0.000} C_DIS
LIN {X 1.743,Y -289.995,Z 88.274,A 90.344,B 90.000,C 0.000} C_DIS
LIN {X 1.776,Y -289.995,Z 88.307,A 90.351,B 90.000,C 0.000} C_DIS
LIN {X 1.842,Y -289.994,Z 88.392,A 90.364,B 90.000,C 0.000} C_DIS
LIN {X 1.928,Y -289.994,Z 88.478,A 90.381,B 90.000,C 0.000} C_DIS
LIN {X 2.013,Y -289.993,Z 88.526,A 90.398,B 90.000,C 0.000} C_DIS
LIN {X 2.923,Y -289.985,Z 89.567,A 90.578,B 90.000,C 0.000} C_DIS
LIN {X 3.009,Y -289.984,Z 89.615,A 90.594,B 90.000,C 0.000} C_DIS
LIN {X 3.094,Y -289.983,Z 89.701,A 90.611,B 90.000,C 0.000} C_DIS
LIN {X 3.147,Y -289.983,Z 89.786,A 90.622,B 90.000,C 0.000} C_DIS
LIN {X 3.235,Y -289.982,Z 89.897,A 90.639,B 90.000,C 0.000} C_DIS
LIN {X 3.468,Y -289.979,Z 90.121,A 90.685,B 90.000,C 0.000} C_DIS
LIN {X 3.552,Y -289.978,Z 90.244,A 90.702,B 90.000,C 0.000} C_DIS
LIN {X 4.118,Y -289.971,Z 90.979,A 90.814,B 90.000,C 0.000} C_DIS
LIN {X 4.178,Y -289.970,Z 91.038,A 90.826,B 90.000,C 0.000} C_DIS
LIN {X 4.402,Y -289.967,Z 91.355,A 90.870,B 90.000,C 0.000} C_DIS
LIN {X 4.680,Y -289.962,Z 91.834,A 90.925,B 90.000,C 0.000} C_DIS
LIN {X 4.784,Y -289.961,Z 92.290,A 90.945,B 90.000,C 0.000} C_DIS
LIN {X 4.798,Y -289.960,Z 92.403,A 90.948,B 90.000,C 0.000} C_DIS
LIN {X 4.904,Y -289.959,Z 92.702,A 90.969,B 90.000,C 0.000} C_DIS
LIN {X 5.261,Y -289.952,Z 94.409,A 91.039,B 90.000,C 0.000} C_DIS
LIN {X 5.304,Y -289.951,Z 94.509,A 91.048,B 90.000,C 0.000} C_DIS
LIN {X 5.329,Y -289.951,Z 94.622,A 91.053,B 90.000,C 0.000} C_DIS
LIN {X 5.410,Y -289.950,Z 94.850,A 91.069,B 90.000,C 0.000} C_DIS
LIN {X 5.535,Y -289.947,Z 95.590,A 91.094,B 90.000,C 0.000} C_DIS
LIN {X 6.099,Y -289.936,Z 98.025,A 91.205,B 90.000,C 0.000} C_DIS
LIN {X 6.228,Y -289.933,Z 98.790,A 91.231,B 90.000,C 0.000} C_DIS
LIN {X 6.280,Y -289.932,Z 98.890,A 91.241,B 90.000,C 0.000} C_DIS
LIN {X 6.377,Y -289.930,Z 99.231,A 91.260,B 90.000,C 0.000} C_DIS
LIN {X 6.392,Y -289.930,Z 99.372,A 91.263,B 90.000,C 0.000} C_DIS
LIN {X 6.861,Y -289.919,Z 101.227,A 91.356,B 90.000,C 0.000} C_DIS
LIN {X 6.873,Y -289.919,Z 101.355,A 91.358,B 90.000,C 0.000} C_DIS
LIN {X 6.946,Y -289.917,Z 101.564,A 91.372,B 90.000,C 0.000} C_DIS
LIN {X 6.956,Y -289.917,Z 101.677,A 91.374,B 90.000,C 0.000} C_DIS
LIN {X 7.253,Y -289.909,Z 102.702,A 91.433,B 90.000,C 0.000} C_DIS
LIN {X 7.263,Y -289.909,Z 102.815,A 91.435,B 90.000,C 0.000} C_DIS
LIN {X 7.401,Y -289.906,Z 103.384,A 91.462,B 90.000,C 0.000} C_DIS
LIN {X 7.416,Y -289.905,Z 103.498,A 91.465,B 90.000,C 0.000} C_DIS
LIN {X 7.488,Y -289.903,Z 103.655,A 91.480,B 90.000,C 0.000} C_DIS
LIN {X 7.978,Y -289.890,Z 106.106,A 91.576,B 90.000,C 0.000} C_DIS
LIN {X 8.496,Y -289.875,Z 108.552,A 91.679,B 90.000,C 0.000} C_DIS
LIN {X 8.635,Y -289.871,Z 109.266,A 91.706,B 90.000,C 0.000} C_DIS
LIN {X 8.710,Y -289.869,Z 109.469,A 91.721,B 90.000,C 0.000} C_DIS
LIN {X 8.720,Y -289.869,Z 109.597,A 91.723,B 90.000,C 0.000} C_DIS
LIN {X 9.204,Y -289.854,Z 111.599,A 91.819,B 90.000,C 0.000} C_DIS
LIN {X 9.339,Y -289.850,Z 112.088,A 91.845,B 90.000,C 0.000} C_DIS
LIN {X 9.354,Y -289.849,Z 112.273,A 91.848,B 90.000,C 0.000} C_DIS
LIN {X 9.879,Y -289.831,Z 114.717,A 91.952,B 90.000,C 0.000} C_DIS
LIN {X 10.385,Y -289.814,Z 117.165,A 92.052,B 90.000,C 0.000} C_DIS
LIN {X 10.618,Y -289.806,Z 118.351,A 92.098,B 90.000,C 0.000} C_DIS
LIN {X 10.756,Y -289.800,Z 118.803,A 92.126,B 90.000,C 0.000} C_DIS
LIN {X 10.770,Y -289.800,Z 118.944,A 92.128,B 90.000,C 0.000} C_DIS
LIN {X 11.003,Y -289.791,Z 119.687,A 92.174,B 90.000,C 0.000} C_DIS
LIN {X 11.039,Y -289.790,Z 119.941,A 92.182,B 90.000,C 0.000} C_DIS
LIN {X 11.690,Y -289.764,Z 122.046,A 92.310,B 90.000,C 0.000} C_DIS
LIN {X 11.699,Y -289.764,Z 122.160,A 92.312,B 90.000,C 0.000} C_DIS
LIN {X 11.721,Y -289.763,Z 122.274,A 92.316,B 90.000,C 0.000} C_DIS
LIN {X 12.033,Y -289.750,Z 123.163,A 92.378,B 90.000,C 0.000} C_DIS
LIN {X 12.319,Y -289.738,Z 124.336,A 92.435,B 90.000,C 0.000} C_DIS
LIN {X 12.368,Y -289.736,Z 124.379,A 92.444,B 90.000,C 0.000} C_DIS
LIN {X 12.395,Y -289.735,Z 124.432,A 92.450,B 90.000,C 0.000} C_DIS
LIN {X 12.412,Y -289.734,Z 124.516,A 92.453,B 90.000,C 0.000} C_DIS
LIN {X 12.663,Y -289.723,Z 125.232,A 92.503,B 90.000,C 0.000} C_DIS
LIN {X 12.708,Y -289.721,Z 125.460,A 92.512,B 90.000,C 0.000} C_DIS
LIN {X 12.951,Y -289.711,Z 126.143,A 92.560,B 90.000,C 0.000} C_DIS
LIN {X 12.992,Y -289.709,Z 126.370,A 92.568,B 90.000,C 0.000} C_DIS
LIN {X 13.161,Y -289.701,Z 126.769,A 92.601,B 90.000,C 0.000} C_DIS
LIN {X 13.201,Y -289.699,Z 126.996,A 92.609,B 90.000,C 0.000} C_DIS
LIN {X 13.453,Y -289.688,Z 127.622,A 92.659,B 90.000,C 0.000} C_DIS
LIN {X 13.492,Y -289.686,Z 127.665,A 92.667,B 90.000,C 0.000} C_DIS
LIN {X 13.727,Y -289.675,Z 128.389,A 92.713,B 90.000,C 0.000} C_DIS
LIN {X 13.785,Y -289.672,Z 128.504,A 92.725,B 90.000,C 0.000} C_DIS
LIN {X 13.908,Y -289.666,Z 128.945,A 92.749,B 90.000,C 0.000} C_DIS
LIN {X 13.949,Y -289.664,Z 128.987,A 92.757,B 90.000,C 0.000} C_DIS
LIN {X 14.183,Y -289.653,Z 129.478,A 92.803,B 90.000,C 0.000} C_DIS
LIN {X 14.524,Y -289.636,Z 130.296,A 92.871,B 90.000,C 0.000} C_DIS
LIN {X 14.553,Y -289.635,Z 130.410,A 92.876,B 90.000,C 0.000} C_DIS
LIN {X 15.035,Y -289.610,Z 131.455,A 92.972,B 90.000,C 0.000} C_DIS
LIN {X 15.096,Y -289.607,Z 131.548,A 92.984,B 90.000,C 0.000} C_DIS
LIN {X 15.146,Y -289.604,Z 131.662,A 92.994,B 90.000,C 0.000} C_DIS
LIN {X 15.266,Y -289.598,Z 131.832,A 93.018,B 90.000,C 0.000} C_DIS
LIN {X 15.316,Y -289.595,Z 131.946,A 93.027,B 90.000,C 0.000} C_DIS
LIN {X 15.376,Y -289.592,Z 132.028,A 93.039,B 90.000,C 0.000} C_DIS
LIN {X 15.774,Y -289.571,Z 132.880,A 93.118,B 90.000,C 0.000} C_DIS
LIN {X 15.888,Y -289.564,Z 133.051,A 93.141,B 90.000,C 0.000} C_DIS
LIN {X 16.456,Y -289.533,Z 134.186,A 93.253,B 90.000,C 0.000} C_DIS
LIN {X 16.516,Y -289.529,Z 134.279,A 93.265,B 90.000,C 0.000} C_DIS
LIN {X 16.566,Y -289.526,Z 134.393,A 93.275,B 90.000,C 0.000} C_DIS
LIN {X 16.686,Y -289.520,Z 134.563,A 93.299,B 90.000,C 0.000} C_DIS
LIN {X 16.730,Y -289.517,Z 134.677,A 93.307,B 90.000,C 0.000} C_DIS
LIN {X 17.548,Y -289.469,Z 135.986,A 93.469,B 90.000,C 0.000} C_DIS
LIN {X 18.770,Y -289.392,Z 137.719,A 93.711,B 90.000,C 0.000} C_DIS
LIN {X 18.841,Y -289.387,Z 137.859,A 93.725,B 90.000,C 0.000} C_DIS
LIN {X 18.982,Y -289.378,Z 138.031,A 93.753,B 90.000,C 0.000} C_DIS
LIN {X 19.132,Y -289.368,Z 138.178,A 93.783,B 90.000,C 0.000} C_DIS
LIN {X 19.219,Y -289.362,Z 138.243,A 93.800,B 90.000,C 0.000} C_DIS
LIN {X 20.823,Y -289.251,Z 140.157,A 94.118,B 90.000,C 0.000} C_DIS
LIN {X 22.489,Y -289.127,Z 142.017,A 94.448,B 90.000,C 0.000} C_DIS
LIN {X 22.700,Y -289.110,Z 142.249,A 94.489,B 90.000,C 0.000} C_DIS
LIN {X 23.013,Y -289.085,Z 142.472,A 94.552,B 90.000,C 0.000} C_DIS
LIN {X 23.295,Y -289.063,Z 142.756,A 94.607,B 90.000,C 0.000} C_DIS
LIN {X 23.380,Y -289.056,Z 142.809,A 94.624,B 90.000,C 0.000} C_DIS
LIN {X 23.495,Y -289.047,Z 142.899,A 94.647,B 90.000,C 0.000} C_DIS
LIN {X 23.576,Y -289.040,Z 142.988,A 94.663,B 90.000,C 0.000} C_DIS
LIN {X 23.598,Y -289.038,Z 143.041,A 94.667,B 90.000,C 0.000} C_DIS
LIN {X 24.466,Y -288.966,Z 143.679,A 94.840,B 90.000,C 0.000} C_DIS
LIN {X 24.571,Y -288.957,Z 143.779,A 94.860,B 90.000,C 0.000} C_DIS
LIN {X 25.591,Y -288.869,Z 144.409,A 95.063,B 90.000,C 0.000} C_DIS
LIN {X 25.931,Y -288.838,Z 144.635,A 95.130,B 90.000,C 0.000} C_DIS
LIN {X 28.201,Y -288.626,Z 145.662,A 95.580,B 90.000,C 0.000} C_DIS
LIN {X 29.089,Y -288.537,Z 145.957,A 95.757,B 90.000,C 0.000} C_DIS
LIN {X 29.161,Y -288.530,Z 145.964,A 95.771,B 90.000,C 0.000} C_DIS
LIN {X 29.206,Y -288.526,Z 145.984,A 95.780,B 90.000,C 0.000} C_DIS
LIN {X 31.639,Y -288.268,Z 146.497,A 96.263,B 90.000,C 0.000} C_DIS
LIN {X 34.075,Y -287.990,Z 146.982,A 96.748,B 90.000,C 0.000} C_DIS
LIN {X 36.521,Y -287.691,Z 147.405,A 97.235,B 90.000,C 0.000} C_DIS
LIN {X 37.910,Y -287.511,Z 147.526,A 97.511,B 90.000,C 0.000} C_DIS
LIN {X 37.984,Y -287.502,Z 147.513,A 97.526,B 90.000,C 0.000} C_DIS
LIN {X 40.455,Y -287.164,Z 147.693,A 98.019,B 90.000,C 0.000} C_DIS
LIN {X 42.594,Y -286.855,Z 147.848,A 98.446,B 90.000,C 0.000} C_DIS
LIN {X 45.063,Y -286.477,Z 147.744,A 98.939,B 90.000,C 0.000} C_DIS
LIN {X 47.515,Y -286.081,Z 147.467,A 99.430,B 90.000,C 0.000} C_DIS
LIN {X 48.159,Y -285.973,Z 147.426,A 99.559,B 90.000,C 0.000} C_DIS
LIN {X 49.218,Y -285.793,Z 147.283,A 99.771,B 90.000,C 0.000} C_DIS
LIN {X 49.561,Y -285.734,Z 147.271,A 99.840,B 90.000,C 0.000} C_DIS
LIN {X 49.743,Y -285.702,Z 147.216,A 99.877,B 90.000,C 0.000} C_DIS
LIN {X 50.962,Y -285.487,Z 147.087,A 100.121,B 90.000,C 0.000} C_DIS
LIN {X 51.039,Y -285.473,Z 147.057,A 100.137,B 90.000,C 0.000} C_DIS
LIN {X 53.261,Y -285.067,Z 146.612,A 100.583,B 90.000,C 0.000} C_DIS
LIN {X 53.387,Y -285.044,Z 146.601,A 100.608,B 90.000,C 0.000} C_DIS
LIN {X 53.480,Y -285.026,Z 146.581,A 100.627,B 90.000,C 0.000} C_DIS
LIN {X 54.207,Y -284.889,Z 146.340,A 100.773,B 90.000,C 0.000} C_DIS
LIN {X 54.319,Y -284.867,Z 146.324,A 100.796,B 90.000,C 0.000} C_DIS
LIN {X 54.538,Y -284.826,Z 146.254,A 100.840,B 90.000,C 0.000} C_DIS
LIN {X 56.822,Y -284.379,Z 145.863,A 101.300,B 90.000,C 0.000} C_DIS
LIN {X 57.891,Y -284.163,Z 145.597,A 101.515,B 90.000,C 0.000} C_DIS
LIN {X 58.458,Y -284.047,Z 145.501,A 101.629,B 90.000,C 0.000} C_DIS
LIN {X 58.885,Y -283.959,Z 145.576,A 101.715,B 90.000,C 0.000} C_DIS
LIN {X 58.983,Y -283.938,Z 145.675,A 101.735,B 90.000,C 0.000} C_DIS
LIN {X 58.985,Y -283.938,Z 145.803,A 101.736,B 90.000,C 0.000} C_DIS
LIN {X 58.998,Y -283.935,Z 145.886,A 101.738,B 90.000,C 0.000} C_DIS
LIN {X 58.961,Y -283.943,Z 148.385,A 101.731,B 90.000,C 0.000} C_DIS
LIN {X 58.925,Y -283.950,Z 148.954,A 101.723,B 90.000,C 0.000} C_DIS
LIN {X 58.977,Y -283.940,Z 149.073,A 101.734,B 90.000,C 0.000} C_DIS
LIN {X 58.869,Y -283.962,Z 150.946,A 101.712,B 90.000,C 0.000} C_DIS
LIN {X 58.916,Y -283.952,Z 151.134,A 101.722,B 90.000,C 0.000} C_DIS
LIN {X 58.812,Y -283.974,Z 152.995,A 101.701,B 90.000,C 0.000} C_DIS
LIN {X 58.863,Y -283.963,Z 153.117,A 101.711,B 90.000,C 0.000} C_DIS
LIN {X 58.766,Y -283.983,Z 155.615,A 101.691,B 90.000,C 0.000} C_DIS
LIN {X 58.701,Y -283.997,Z 158.114,A 101.678,B 90.000,C 0.000} C_DIS
LIN {X 58.637,Y -284.010,Z 160.613,A 101.665,B 90.000,C 0.000} C_DIS
LIN {X 58.554,Y -284.027,Z 163.111,A 101.649,B 90.000,C 0.000} C_DIS
LIN {X 58.536,Y -284.031,Z 163.454,A 101.645,B 90.000,C 0.000} C_DIS
LIN {X 58.560,Y -284.026,Z 163.580,A 101.650,B 90.000,C 0.000} C_DIS
LIN {X 58.584,Y -284.021,Z 163.645,A 101.655,B 90.000,C 0.000} C_DIS
LIN {X 58.484,Y -284.042,Z 166.142,A 101.635,B 90.000,C 0.000} C_DIS
LIN {X 58.427,Y -284.053,Z 167.492,A 101.623,B 90.000,C 0.000} C_DIS
LIN {X 58.455,Y -284.047,Z 167.620,A 101.629,B 90.000,C 0.000} C_DIS
LIN {X 58.475,Y -284.043,Z 167.679,A 101.633,B 90.000,C 0.000} C_DIS
LIN {X 58.367,Y -284.066,Z 169.495,A 101.611,B 90.000,C 0.000} C_DIS
LIN {X 58.394,Y -284.060,Z 169.554,A 101.616,B 90.000,C 0.000} C_DIS
LIN {X 58.418,Y -284.055,Z 169.678,A 101.621,B 90.000,C 0.000} C_DIS
LIN {X 58.314,Y -284.077,Z 171.482,A 101.600,B 90.000,C 0.000} C_DIS
LIN {X 58.363,Y -284.067,Z 171.607,A 101.610,B 90.000,C 0.000} C_DIS
LIN {X 58.267,Y -284.086,Z 174.105,A 101.591,B 90.000,C 0.000} C_DIS
LIN {X 58.203,Y -284.099,Z 176.604,A 101.578,B 90.000,C 0.000} C_DIS
LIN {X 58.133,Y -284.114,Z 179.103,A 101.564,B 90.000,C 0.000} C_DIS
LIN {X 58.062,Y -284.128,Z 181.602,A 101.550,B 90.000,C 0.000} C_DIS
LIN {X 57.993,Y -284.142,Z 184.100,A 101.536,B 90.000,C 0.000} C_DIS
LIN {X 57.922,Y -284.157,Z 186.599,A 101.521,B 90.000,C 0.000} C_DIS
LIN {X 57.868,Y -284.168,Z 187.413,A 101.510,B 90.000,C 0.000} C_DIS
LIN {X 57.894,Y -284.162,Z 187.476,A 101.516,B 90.000,C 0.000} C_DIS
LIN {X 57.919,Y -284.157,Z 187.633,A 101.521,B 90.000,C 0.000} C_DIS
LIN {X 57.812,Y -284.179,Z 189.399,A 101.499,B 90.000,C 0.000} C_DIS
LIN {X 57.777,Y -284.186,Z 191.506,A 101.492,B 90.000,C 0.000} C_DIS
LIN {X 57.800,Y -284.181,Z 191.585,A 101.497,B 90.000,C 0.000} C_DIS
LIN {X 57.698,Y -284.202,Z 194.083,A 101.476,B 90.000,C 0.000} C_DIS
LIN {X 57.603,Y -284.222,Z 196.581,A 101.457,B 90.000,C 0.000} C_DIS
LIN {X 57.589,Y -284.224,Z 196.795,A 101.454,B 90.000,C 0.000} C_DIS
LIN {X 57.612,Y -284.220,Z 196.921,A 101.459,B 90.000,C 0.000} C_DIS
LIN {X 57.636,Y -284.215,Z 196.985,A 101.464,B 90.000,C 0.000} C_DIS
LIN {X 57.529,Y -284.237,Z 199.482,A 101.442,B 90.000,C 0.000} C_DIS
LIN {X 57.477,Y -284.247,Z 200.215,A 101.432,B 90.000,C 0.000} C_DIS
LIN {X 57.521,Y -284.238,Z 200.406,A 101.440,B 90.000,C 0.000} C_DIS
LIN {X 57.397,Y -284.263,Z 202.903,A 101.415,B 90.000,C 0.000} C_DIS
LIN {X 57.362,Y -284.270,Z 203.691,A 101.408,B 90.000,C 0.000} C_DIS
LIN {X 57.413,Y -284.260,Z 203.812,A 101.419,B 90.000,C 0.000} C_DIS
LIN {X 57.301,Y -284.283,Z 206.310,A 101.396,B 90.000,C 0.000} C_DIS
LIN {X 57.195,Y -284.304,Z 208.526,A 101.375,B 90.000,C 0.000} C_DIS
LIN {X 57.212,Y -284.301,Z 208.585,A 101.378,B 90.000,C 0.000} C_DIS
LIN {X 57.181,Y -284.307,Z 209.664,A 101.372,B 90.000,C 0.000} C_DIS
LIN {X 57.042,Y -284.335,Z 209.958,A 101.344,B 90.000,C 0.000} C_DIS
LIN {X 56.411,Y -284.461,Z 210.034,A 101.217,B 90.000,C 0.000} C_DIS
LIN {X 54.831,Y -284.769,Z 210.007,A 100.899,B 90.000,C 0.000} C_DIS
LIN {X 54.754,Y -284.784,Z 210.028,A 100.883,B 90.000,C 0.000} C_DIS
LIN {X 52.300,Y -285.245,Z 209.905,A 100.390,B 90.000,C 0.000} C_DIS
LIN {X 49.864,Y -285.681,Z 209.554,A 99.901,B 90.000,C 0.000} C_DIS
LIN {X 47.472,Y -286.088,Z 208.952,A 99.421,B 90.000,C 0.000} C_DIS
LIN {X 45.103,Y -286.471,Z 208.250,A 98.947,B 90.000,C 0.000} C_DIS
LIN {X 44.115,Y -286.625,Z 207.850,A 98.750,B 90.000,C 0.000} C_DIS
LIN {X 43.552,Y -286.711,Z 207.727,A 98.637,B 90.000,C 0.000} C_DIS
LIN {X 41.223,Y -287.055,Z 206.887,A 98.172,B 90.000,C 0.000} C_DIS
LIN {X 38.914,Y -287.377,Z 205.985,A 97.712,B 90.000,C 0.000} C_DIS
LIN {X 36.597,Y -287.682,Z 205.097,A 97.250,B 90.000,C 0.000} C_DIS
LIN {X 35.379,Y -287.834,Z 204.488,A 97.007,B 90.000,C 0.000} C_DIS
LIN {X 35.053,Y -287.874,Z 204.282,A 96.943,B 90.000,C 0.000} C_DIS
LIN {X 34.865,Y -287.897,Z 204.204,A 96.905,B 90.000,C 0.000} C_DIS
LIN {X 34.587,Y -287.930,Z 204.033,A 96.850,B 90.000,C 0.000} C_DIS
LIN {X 34.406,Y -287.952,Z 203.955,A 96.814,B 90.000,C 0.000} C_DIS
LIN {X 34.080,Y -287.991,Z 203.749,A 96.749,B 90.000,C 0.000} C_DIS
LIN {X 33.741,Y -288.030,Z 203.577,A 96.681,B 90.000,C 0.000} C_DIS
LIN {X 33.415,Y -288.068,Z 203.371,A 96.617,B 90.000,C 0.000} C_DIS
LIN {X 33.235,Y -288.089,Z 203.294,A 96.581,B 90.000,C 0.000} C_DIS
LIN {X 32.837,Y -288.135,Z 203.063,A 96.502,B 90.000,C 0.000} C_DIS
LIN {X 32.418,Y -288.182,Z 202.781,A 96.418,B 90.000,C 0.000} C_DIS
LIN {X 32.319,Y -288.194,Z 202.739,A 96.399,B 90.000,C 0.000} C_DIS
LIN {X 30.622,Y -288.379,Z 201.473,A 96.061,B 90.000,C 0.000} C_DIS
LIN {X 30.603,Y -288.381,Z 201.416,A 96.058,B 90.000,C 0.000} C_DIS
LIN {X 30.548,Y -288.387,Z 201.359,A 96.047,B 90.000,C 0.000} C_DIS
LIN {X 30.425,Y -288.400,Z 201.274,A 96.022,B 90.000,C 0.000} C_DIS
LIN {X 30.342,Y -288.408,Z 201.188,A 96.006,B 90.000,C 0.000} C_DIS
LIN {X 29.792,Y -288.466,Z 200.733,A 95.896,B 90.000,C 0.000} C_DIS
LIN {X 29.544,Y -288.491,Z 200.449,A 95.847,B 90.000,C 0.000} C_DIS
LIN {X 28.948,Y -288.552,Z 199.960,A 95.729,B 90.000,C 0.000} C_DIS
LIN {X 28.885,Y -288.558,Z 199.817,A 95.716,B 90.000,C 0.000} C_DIS
LIN {X 28.723,Y -288.574,Z 199.709,A 95.684,B 90.000,C 0.000} C_DIS
LIN {X 28.590,Y -288.587,Z 199.538,A 95.658,B 90.000,C 0.000} C_DIS
LIN {X 28.084,Y -288.637,Z 199.030,A 95.557,B 90.000,C 0.000} C_DIS
LIN {X 27.706,Y -288.673,Z 198.685,A 95.482,B 90.000,C 0.000} C_DIS
LIN {X 27.631,Y -288.681,Z 198.640,A 95.467,B 90.000,C 0.000} C_DIS
LIN {X 26.271,Y -288.808,Z 197.033,A 95.198,B 90.000,C 0.000} C_DIS
LIN {X 24.798,Y -288.938,Z 195.214,A 94.905,B 90.000,C 0.000} C_DIS
LIN {X 24.738,Y -288.943,Z 195.157,A 94.893,B 90.000,C 0.000} C_DIS
LIN {X 24.710,Y -288.945,Z 195.105,A 94.888,B 90.000,C 0.000} C_DIS
LIN {X 24.629,Y -288.952,Z 195.015,A 94.872,B 90.000,C 0.000} C_DIS
LIN {X 24.514,Y -288.962,Z 194.935,A 94.849,B 90.000,C 0.000} C_DIS
LIN {X 24.231,Y -288.986,Z 194.517,A 94.793,B 90.000,C 0.000} C_DIS
LIN {X 24.146,Y -288.993,Z 194.475,A 94.776,B 90.000,C 0.000} C_DIS
LIN {X 24.061,Y -289.000,Z 194.389,A 94.759,B 90.000,C 0.000} C_DIS
LIN {X 24.001,Y -289.005,Z 194.304,A 94.747,B 90.000,C 0.000} C_DIS
LIN {X 23.976,Y -289.007,Z 194.247,A 94.742,B 90.000,C 0.000} C_DIS
LIN {X 23.960,Y -289.009,Z 194.190,A 94.739,B 90.000,C 0.000} C_DIS
LIN {X 23.642,Y -289.035,Z 193.792,A 94.676,B 90.000,C 0.000} C_DIS
LIN {X 22.951,Y -289.090,Z 192.583,A 94.539,B 90.000,C 0.000} C_DIS
LIN {X 22.529,Y -289.124,Z 191.828,A 94.456,B 90.000,C 0.000} C_DIS
LIN {X 22.485,Y -289.127,Z 191.687,A 94.447,B 90.000,C 0.000} C_DIS
LIN {X 22.371,Y -289.136,Z 191.559,A 94.424,B 90.000,C 0.000} C_DIS
LIN {X 22.139,Y -289.154,Z 191.137,A 94.378,B 90.000,C 0.000} C_DIS
LIN {X 22.005,Y -289.164,Z 190.810,A 94.352,B 90.000,C 0.000} C_DIS
LIN {X 21.662,Y -289.190,Z 190.378,A 94.284,B 90.000,C 0.000} C_DIS
LIN {X 21.338,Y -289.214,Z 189.663,A 94.220,B 90.000,C 0.000} C_DIS
LIN {X 21.224,Y -289.222,Z 189.482,A 94.197,B 90.000,C 0.000} C_DIS
LIN {X 20.998,Y -289.239,Z 188.942,A 94.152,B 90.000,C 0.000} C_DIS
LIN {X 20.907,Y -289.245,Z 188.794,A 94.134,B 90.000,C 0.000} C_DIS
LIN {X 20.709,Y -289.260,Z 188.330,A 94.095,B 90.000,C 0.000} C_DIS
LIN {X 20.657,Y -289.263,Z 188.249,A 94.085,B 90.000,C 0.000} C_DIS
LIN {X 20.366,Y -289.284,Z 187.647,A 94.027,B 90.000,C 0.000} C_DIS
LIN {X 20.327,Y -289.287,Z 187.533,A 94.019,B 90.000,C 0.000} C_DIS
LIN {X 19.794,Y -289.324,Z 186.324,A 93.914,B 90.000,C 0.000} C_DIS
LIN {X 19.749,Y -289.327,Z 186.282,A 93.905,B 90.000,C 0.000} C_DIS
LIN {X 19.692,Y -289.331,Z 186.200,A 93.894,B 90.000,C 0.000} C_DIS
LIN {X 19.232,Y -289.362,Z 185.314,A 93.803,B 90.000,C 0.000} C_DIS
LIN {X 19.104,Y -289.370,Z 185.017,A 93.777,B 90.000,C 0.000} C_DIS
LIN {X 18.897,Y -289.384,Z 184.689,A 93.736,B 90.000,C 0.000} C_DIS
LIN {X 18.844,Y -289.387,Z 184.461,A 93.726,B 90.000,C 0.000} C_DIS
LIN {X 18.613,Y -289.402,Z 184.077,A 93.680,B 90.000,C 0.000} C_DIS
LIN {X 17.902,Y -289.447,Z 182.474,A 93.539,B 90.000,C 0.000} C_DIS
LIN {X 17.883,Y -289.448,Z 182.389,A 93.535,B 90.000,C 0.000} C_DIS
LIN {X 17.308,Y -289.483,Z 180.307,A 93.422,B 90.000,C 0.000} C_DIS
LIN {X 17.256,Y -289.486,Z 180.194,A 93.411,B 90.000,C 0.000} C_DIS
LIN {X 17.237,Y -289.487,Z 180.071,A 93.407,B 90.000,C 0.000} C_DIS
LIN {X 16.907,Y -289.507,Z 179.056,A 93.342,B 90.000,C 0.000} C_DIS
LIN {X 16.894,Y -289.508,Z 178.942,A 93.340,B 90.000,C 0.000} C_DIS
LIN {X 16.856,Y -289.510,Z 178.828,A 93.332,B 90.000,C 0.000} C_DIS
LIN {X 16.802,Y -289.513,Z 178.729,A 93.321,B 90.000,C 0.000} C_DIS
LIN {X 16.539,Y -289.528,Z 177.181,A 93.269,B 90.000,C 0.000} C_DIS
LIN {X 16.437,Y -289.534,Z 176.837,A 93.249,B 90.000,C 0.000} C_DIS
LIN {X 15.930,Y -289.562,Z 174.389,A 93.149,B 90.000,C 0.000} C_DIS
LIN {X 15.488,Y -289.586,Z 171.929,A 93.061,B 90.000,C 0.000} C_DIS
LIN {X 14.991,Y -289.612,Z 169.479,A 92.963,B 90.000,C 0.000} C_DIS
LIN {X 14.533,Y -289.636,Z 167.021,A 92.872,B 90.000,C 0.000} C_DIS
LIN {X 14.213,Y -289.651,Z 165.227,A 92.809,B 90.000,C 0.000} C_DIS
LIN {X 14.180,Y -289.653,Z 165.163,A 92.803,B 90.000,C 0.000} C_DIS
LIN {X 14.051,Y -289.659,Z 164.548,A 92.777,B 90.000,C 0.000} C_DIS
LIN {X 13.845,Y -289.669,Z 162.056,A 92.736,B 90.000,C 0.000} C_DIS
LIN {X 13.765,Y -289.673,Z 160.721,A 92.721,B 90.000,C 0.000} C_DIS
LIN {X 13.553,Y -289.683,Z 158.230,A 92.679,B 90.000,C 0.000} C_DIS
LIN {X 13.366,Y -289.692,Z 155.737,A 92.642,B 90.000,C 0.000} C_DIS
LIN {X 13.297,Y -289.695,Z 155.373,A 92.628,B 90.000,C 0.000} C_DIS
LIN {X 13.137,Y -289.702,Z 153.524,A 92.596,B 90.000,C 0.000} C_DIS
LIN {X 13.083,Y -289.705,Z 153.339,A 92.586,B 90.000,C 0.000} C_DIS
LIN {X 13.063,Y -289.706,Z 152.941,A 92.582,B 90.000,C 0.000} C_DIS
LIN {X 13.012,Y -289.708,Z 152.756,A 92.572,B 90.000,C 0.000} C_DIS
LIN {X 12.908,Y -289.713,Z 151.866,A 92.551,B 90.000,C 0.000} C_DIS
LIN {X 12.909,Y -289.713,Z 151.663,A 92.551,B 90.000,C 0.000} C_DIS
LIN {X 12.884,Y -289.714,Z 151.518,A 92.546,B 90.000,C 0.000} C_DIS
LIN {X 12.851,Y -289.715,Z 151.444,A 92.540,B 90.000,C 0.000} C_DIS
LIN {X 12.744,Y -289.720,Z 150.216,A 92.519,B 90.000,C 0.000} C_DIS
LIN {X 12.657,Y -289.724,Z 149.754,A 92.502,B 90.000,C 0.000} C_DIS
LIN {X 12.625,Y -289.725,Z 149.677,A 92.495,B 90.000,C 0.000} C_DIS
LIN {X 12.460,Y -289.732,Z 148.389,A 92.462,B 90.000,C 0.000} C_DIS
LIN {X 12.496,Y -289.731,Z 147.991,A 92.470,B 90.000,C 0.000} C_DIS
LIN {X 12.584,Y -289.727,Z 147.722,A 92.487,B 90.000,C 0.000} C_DIS
LIN {X 12.754,Y -289.719,Z 147.693,A 92.521,B 90.000,C 0.000} C_DIS
LIN {X 12.983,Y -289.709,Z 147.778,A 92.566,B 90.000,C 0.000} C_DIS
LIN {X 13.283,Y -289.696,Z 148.095,A 92.625,B 90.000,C 0.000} C_DIS
LIN {X 13.345,Y -289.693,Z 148.242,A 92.637,B 90.000,C 0.000} C_DIS
LIN {X 13.378,Y -289.691,Z 148.275,A 92.644,B 90.000,C 0.000} C_DIS
LIN {X 13.501,Y -289.686,Z 148.503,A 92.668,B 90.000,C 0.000} C_DIS
LIN {X 13.558,Y -289.683,Z 148.579,A 92.680,B 90.000,C 0.000} C_DIS
